# B&R Automation Studio project Panasonic_LinkaPowerCP2_A2021055 (part 30)

#### Main.st - Init, cyclic, exit code
```iecst
PROGRAM _INIT
	(* Insert code here *)

END_PROGRAM

PROGRAM _CYCLIC

	//**********************************************************IO modul Wedmuller**********************************************************************//
	//************Karta AB 3.5 8DI**************//
	P3_Pracovisko.IN.StavPrepatovejOchrany_OK := P3_Pracovisko.COM_Weidmuller.AB3_5_8DI.0;
	P3_Srobovanie.IN.NapajanieSkrutkovackyK40_OK := P3_Pracovisko.COM_Weidmuller.AB3_5_8DI.1;
	P3_Srobovanie.IN.NapajanieSkrutkovackyM5_OK := P3_Pracovisko.COM_Weidmuller.AB3_5_8DI.2;
	P3_Srobovanie.IN.NapajanieZasobnikaK40_OK := P3_Pracovisko.COM_Weidmuller.AB3_5_8DI.3;
	P3_Srobovanie.IN.NapajanieZasobnikaM5_OK := P3_Pracovisko.COM_Weidmuller.AB3_5_8DI.4;
	P3_Srobovanie.IN.NapajanieVibrolistyM5_OK := P3_Pracovisko.COM_Weidmuller.AB3_5_8DI.5;
	P3_LeakageTestA.IN.NapajanieTestera_OK := P3_Pracovisko.COM_Weidmuller.AB3_5_8DI.6;
	P3_LeakageTestB.IN.NapajanieTestera_OK := P3_Pracovisko.COM_Weidmuller.AB3_5_8DI.7;

	//************Karta AB 3.6 8DI**************//
	P3_Dopravniky.IN.StavRiadPredDopravBunky_READY := P3_Pracovisko.COM_Weidmuller.AB3_6_8DI.0;
	P3_Dopravniky.IN.StavRiadeniaPriecnDoprav1_READY := P3_Pracovisko.COM_Weidmuller.AB3_6_8DI.1;
	P3_Dopravniky.IN.StavRiadeniaPriecnDoprav2_READY := P3_Pracovisko.COM_Weidmuller.AB3_6_8DI.2;
	P3_Dopravniky.IN.StavRiadZadnDopravBunky_READY := P3_Pracovisko.COM_Weidmuller.AB3_6_8DI.3;
	P3_Dopravniky.IN.StavRiadeniaVratnehoDoprav_READY := P3_Pracovisko.COM_Weidmuller.AB3_6_8DI.4;
	P3_Dopravniky.IN.TeplotaMotoraPredDopravBunky_OK := P3_Pracovisko.COM_Weidmuller.AB3_6_8DI.5;
	P3_Dopravniky.IN.TeplotaMotoraPriecnDoprav1_OK := P3_Pracovisko.COM_Weidmuller.AB3_6_8DI.6;
	P3_Dopravniky.IN.TeplotaMotoraPriecnDoprav2_OK := P3_Pracovisko.COM_Weidmuller.AB3_6_8DI.7;

	//************Karta AB 3.7 8DI**************//
	P3_Dopravniky.IN.TeplotaMotoraZadnDopravBunky_OK := P3_Pracovisko.COM_Weidmuller.AB3_7_8DI.0;
	P3_Dopravniky.IN.TeplotaMotoraVratnehoDoprav_OK := P3_Pracovisko.COM_Weidmuller.AB3_7_8DI.1;
	P3_Pracovisko.COM_Weidmuller.AB3_7_8DI.2;
	P3_Pracovisko.COM_Weidmuller.AB3_7_8DI.3;
	Safety.IN.Linka_SV_ZonaCS := P3_Pracovisko.COM_Weidmuller.AB3_7_8DI.4;
	Safety.IN.P3_SV_ZonaBunky := P3_Pracovisko.COM_Weidmuller.AB3_7_8DI.5;
	Safety.IN.P3_SV_HV_test := P3_Pracovisko.COM_Weidmuller.AB3_7_8DI.6;
	P3_Pracovisko.COM_Weidmuller.AB3_7_8DI.7;

	//************Karta AB 3.8 8DI**************//
	P3_Pracovisko.COM_Weidmuller.AB3_8_8DI.0;
	P3_Pracovisko.COM_Weidmuller.AB3_8_8DI.1;
	P3_Pracovisko.COM_Weidmuller.AB3_8_8DI.2;
	P3_Pracovisko.COM_Weidmuller.AB3_8_8DI.3;
	P3_Pracovisko.COM_Weidmuller.AB3_8_8DI.4;
	P3_Pracovisko.COM_Weidmuller.AB3_8_8DI.5;
	P3_Pracovisko.COM_Weidmuller.AB3_8_8DI.6;
	P3_Pracovisko.COM_Weidmuller.AB3_8_8DI.7;

	//************Karta AB 3.9 8DO***************//
	P3_Pracovisko.COM_Weidmuller.AB3_9_8DO.0 := P3_Pracovisko.OUT.Majak_ZeleneSvetlo_ON;
	P3_Pracovisko.COM_Weidmuller.AB3_9_8DO.1 := P3_Pracovisko.OUT.Majak_OranzoveSvetlo_ON;
	P3_Pracovisko.COM_Weidmuller.AB3_9_8DO.2 := P3_Pracovisko.OUT.Majak_CerveneSvetlo_ON;
	P3_Pracovisko.COM_Weidmuller.AB3_9_8DO.3 := P3_Pracovisko.OUT.Majak_Hukacka_ON;
	P3_Pracovisko.COM_Weidmuller.AB3_9_8DO.4 := P3_Srobovanie.SkrutSet_K40.OUT.VibracnyHrniec.ZapniVibromotor;
	P3_Pracovisko.COM_Weidmuller.AB3_9_8DO.5 := P3_Srobovanie.SkrutSet_M5.OUT.VibropohonZasobnika_RUN;
	P3_Pracovisko.COM_Weidmuller.AB3_9_8DO.6 := P3_Srobovanie.SkrutSet_M5.OUT.VibropohonListy_RUN;
	P3_Pracovisko.COM_Weidmuller.AB3_9_8DO.7 := P3_Pracovisko.OUT.OsvetlenieBunky_ON;

	//************Karta AB 3.10 8DO***************//
	P3_Pracovisko.COM_Weidmuller.AB3_10_8DO.0;
	P3_Pracovisko.COM_Weidmuller.AB3_10_8DO.1;
	P3_Pracovisko.COM_Weidmuller.AB3_10_8DO.2;
	P3_Pracovisko.COM_Weidmuller.AB3_10_8DO.3;
	P3_Pracovisko.COM_Weidmuller.AB3_10_8DO.4;
	P3_Pracovisko.COM_Weidmuller.AB3_10_8DO.5:= Safety.OUT.Linka_ResetCS;
	P3_Pracovisko.COM_Weidmuller.AB3_10_8DO.6:= Safety.OUT.P3_ResetZonyBunky;
	P3_Pracovisko.COM_Weidmuller.AB3_10_8DO.7:= Safety.OUT.P3_ResetZonyHVtest;

	P3_Pracovisko.COM_Weidmuller.AB3_10_8DO.0 := P3_Dopravniky.OUT.PrednyDopravnikBunky_ON;
	P3_Pracovisko.COM_Weidmuller.AB3_10_8DO.1 := P3_Dopravniky.OUT.PriecnyDopravnik1_VPRED;
	P3_Pracovisko.COM_Weidmuller.AB3_10_8DO.2 := P3_Dopravniky.OUT.PriecnyDopravnik2_VPRED;
	P3_Pracovisko.COM_Weidmuller.AB3_10_8DO.3 := P3_Dopravniky.OUT.ZadnyDopravnikBunky_ON;
	P3_Pracovisko.COM_Weidmuller.AB3_10_8DO.4 := P3_Dopravniky.OUT.VratnyDopravnik_ON;
	P3_Pracovisko.COM_Weidmuller.AB3_10_8DO.5;
	P3_Pracovisko.COM_Weidmuller.AB3_10_8DO.6;
	P3_Pracovisko.COM_Weidmuller.AB3_10_8DO.7;

	//************Karta AB 3.12 8DO***************//
	P3_Pracovisko.COM_Weidmuller.AB3_12_8DO.0;
	P3_Pracovisko.COM_Weidmuller.AB3_12_8DO.1;
	P3_Pracovisko.COM_Weidmuller.AB3_12_8DO.2;
	P3_Pracovisko.COM_Weidmuller.AB3_12_8DO.3;
	P3_Pracovisko.COM_Weidmuller.AB3_12_8DO.4;
	P3_Pracovisko.COM_Weidmuller.AB3_12_8DO.5;
	P3_Pracovisko.COM_Weidmuller.AB3_12_8DO.6 := P3_Dopravniky.OUT.PriecnyDopravnik2_VZAD;
	P3_Pracovisko.COM_Weidmuller.AB3_12_8DO.7 := P3_Pracovisko.OUT.Ventilator_ON;

	//**************************************************************IO modul Festo**********************************************************************************//

	//**********Modul DM 3.1 4DI4DO**************//
	//Inputs//
	P3_Pracovisko.IN.PredneDvereLave_PritomnAdaptera := P3_Pracovisko.COM_Festo.DM3_1_4DI[0];
	P3_Pracovisko.IN.PredneDverePrave_PritomnAdaptera := P3_Pracovisko.COM_Festo.DM3_1_4DI[1];
	P3_Pracovisko.IN.ZadneDvereLave_PritomnAdaptera := P3_Pracovisko.COM_Festo.DM3_1_4DI[2];
	P3_Pracovisko.IN.ZadneDverePrave_PritomnAdaptera := P3_Pracovisko.COM_Festo.DM3_1_4DI[3];

	//Outputs//
	P3_Pracovisko.COM_Festo.DM3_1_4DO[0] := P3_Pracovisko.OUT.PredneDvereLave_ZAMKNI;
	P3_Pracovisko.COM_Festo.DM3_1_4DO[1] := P3_Pracovisko.OUT.PredneDverePrave_ZAMKNI;
	P3_Pracovisko.COM_Festo.DM3_1_4DO[2] := P3_Pracovisko.OUT.ZadneDvereLave_ZAMKNI;
	P3_Pracovisko.COM_Festo.DM3_1_4DO[3] := P3_Pracovisko.OUT.ZadneDverePrave_ZAMKNI;

	//***********Modul DI 3.1 8DI****************//
	P3_HV_Test.IN.HorneKontakty_VYSUNUTE := P3_Pracovisko.COM_Festo.DI3_1_8DI[0];
	P3_HV_Test.IN.HorneKontakty_ZASUNUTE := P3_Pracovisko.COM_Festo.DI3_1_8DI[1];
	P3_HV_Test.IN.Centrovanie_ZASUNUTE := P3_Pracovisko.COM_Festo.DI3_1_8DI[2];
	P3_HV_Test.IN.Centrovanie_VYSUNUTE := P3_Pracovisko.COM_Festo.DI3_1_8DI[3];
	P3_HV_Test.IN.SpodneKontakty_ZASUNUTE := P3_Pracovisko.COM_Festo.DI3_1_8DI[4];
	P3_HV_Test.IN.SpodneKontakty_VYSUNUTE := P3_Pracovisko.COM_Festo.DI3_1_8DI[5];
	P3_HV_Test.IN.TypKonektoru_5F_5H := P3_Pracovisko.COM_Festo.DI3_1_8DI[6];
	P3_HV_Test.IN.TypKonektoru_4F := P3_Pracovisko.COM_Festo.DI3_1_8DI[7];

	//***********Modul DI 3.2 8DI****************//
	P3_Pracovisko.COM_Festo.DI3_2_8DI[0];
	P3_ZdvizkaZaLeakTestA.IN.TlmicPaletky_ZASUNUTY := P3_Pracovisko.COM_Festo.DI3_2_8DI[1];
	P3_ZdvizkaZaLeakTestB.IN.TlmicPaletky_ZASUNUTY := P3_Pracovisko.COM_Festo.DI3_2_8DI[2];
	P3_Pracovisko.COM_Festo.DI3_2_8DI[3];
	P3_Pracovisko.COM_Festo.DI3_2_8DI[4];
	P3_Pracovisko.COM_Festo.DI3_2_8DI[5];
	P3_Pracovisko.COM_Festo.DI3_2_8DI[6];
	P3_Pracovisko.COM_Festo.DI3_2_8DI[7];

	//***********Modul DI 3.3 8DI****************//
	P3_LeakageTestA.IN.HornyPritlak_TlakOK := P3_Pracovisko.COM_Festo.DI3_4_8DI[0];
	P3_LeakageTestA.IN.HornyPritlak_PneuZamok_Odomknuty := P3_Pracovisko.COM_Festo.DI3_4_8DI[1];
	P3_LeakageTestB.IN.HornyPritlak_ZASUNUTY := P3_Pracovisko.COM_Festo.DI3_3_8DI[2];
	P3_LeakageTestB.IN.HornyPritlak_VYSUNUTY := P3_Pracovisko.COM_Festo.DI3_3_8DI[3];
	P3_LeakageTestB.IN.PritomnostKopita := P3_Pracovisko.COM_Festo.DI3_3_8DI[4];
	P3_LeakageTestB.IN.Kopito_ZASUNUTE := P3_Pracovisko.COM_Festo.DI3_3_8DI[5];
	P3_LeakageTestB.IN.Centrovanie_VYSUNUTE := P3_Pracovisko.COM_Festo.DI3_3_8DI[6];
	P3_LeakageTestB.IN.Centrovanie_ZASUNUTE := P3_Pracovisko.COM_Festo.DI3_3_8DI[7];

	//***********Modul DI 3.4 8DI****************//
	P3_LeakageTestB.IN.HornyPritlak_TlakOK:= P3_Pracovisko.COM_Festo.DI3_3_8DI[0];
	P3_LeakageTestB.IN.HornyPritlak_PneuZamok_Odomknuty := P3_Pracovisko.COM_Festo.DI3_3_8DI[1];
	P3_LeakageTestA.IN.HornyPritlak_VYSUNUTY := P3_Pracovisko.COM_Festo.DI3_4_8DI[2];
	P3_LeakageTestA.IN.HornyPritlak_ZASUNUTY := P3_Pracovisko.COM_Festo.DI3_4_8DI[3];
	P3_LeakageTestA.IN.PritomnostKopita := P3_Pracovisko.COM_Festo.DI3_4_8DI[4];
	P3_LeakageTestA.IN.Kopito_ZASUNUTE := P3_Pracovisko.COM_Festo.DI3_4_8DI[5];
	P3_LeakageTestA.IN.Centrovanie_VYSUNUTE := P3_Pracovisko.COM_Festo.DI3_4_8DI[6];
	P3_LeakageTestA.IN.Centrovanie_ZASUNUTE := P3_Pracovisko.COM_Festo.DI3_4_8DI[7];

	//***********Modul DI 3.5 8DI****************//
	P3_Srobovanie.SkrutSet_K40.IN.VibracnyHrniec.PritomnostSkrutiekVHrnci := P3_Pracovisko.COM_Festo.DI3_5_8DI[0];
	P3_Srobovanie.SkrutSet_K40.IN.VibracnyHrniec.VibracnaListaZaplnena := P3_Pracovisko.COM_Festo.DI3_5_8DI[1];
	P3_Srobovanie.SkrutSet_K40.IN.VibracnyHrniec.PreletovySnimac := P3_Pracovisko.COM_Festo.DI3_5_8DI[2];
	P3_Srobovanie.SkrutSet_K40.IN.Brzda.PodajSkrutku:= P3_Pracovisko.COM_Festo.DI3_5_8DI[3];
	P3_Srobovanie.SkrutSet_K40.IN.Brzda.ZakladnaPoloha  := P3_Pracovisko.COM_Festo.DI3_5_8DI[4];
	P3_Srobovanie.SkrutSet_K40.IN.Brzda.SkrutkaPritomnaVBrzde := P3_Pracovisko.COM_Festo.DI3_5_8DI[5];
	P3_Srobovanie.SkrutSet_K40.IN.Brzda.PreletSkrutky := P3_Pracovisko.COM_Festo.DI3_5_8DI[6];
	P3_Srobovanie.IN.Skrutkovacka_K40_ZASUNUTA := P3_Pracovisko.COM_Festo.DI3_5_8DI[7];

	//***********Modul DI 3.6 8DI****************//
	P3_Srobovanie.SkrutSet_M5.IN.ZasobnikSkrutiekPrazdny := P3_Pracovisko.COM_Festo.DI3_6_8DI[0];
	P3_Srobovanie.SkrutSet_M5.IN.ZaplnenieListyZasobnika := P3_Pracovisko.COM_Festo.DI3_6_8DI[1];
	P3_Srobovanie.SkrutSet_M5.IN.ZaplnenieVibrolisty_MAX := P3_Pracovisko.COM_Festo.DI3_6_8DI[2];
	P3_Srobovanie.SkrutSet_M5.IN.ZaplnenieVibrolisty_MIN := P3_Pracovisko.COM_Festo.DI3_6_8DI[3];
	P3_Srobovanie.SkrutSet_M5.IN.Podavac_SkrutkaNaVstupe := P3_Pracovisko.COM_Festo.DI3_6_8DI[4];
	P3_Srobovanie.SkrutSet_M5.IN.Podavac_SkrutkaNaVystupe := P3_Pracovisko.COM_Festo.DI3_6_8DI[5];
	P3_Srobovanie.SkrutSet_M5.IN.PodavacOtoceny_VSTUP := P3_Pracovisko.COM_Festo.DI3_6_8DI[6];
	P3_Srobovanie.SkrutSet_M5.IN.PodavacOtoceny_VYSTUP := P3_Pracovisko.COM_Festo.DI3_6_8DI[7];

	//***********Modul DI 3.7 8DI****************//
	P3_Srobovanie.IN.Skrutkovacka_M5_Vakum_OK := P3_Pracovisko.COM_Festo.DI3_7_8DI[0];
	P3_Pracovisko.IN.TlakVzduchu_OK := P3_Pracovisko.COM_Festo.DI3_7_8DI[1];
	Safety.IN.P3_SV_PrivodVzduchu_CH1 := P3_Pracovisko.COM_Festo.DI3_7_8DI[2];
	Safety.IN.P3_SV_PrivodVzduchu_CH2 := P3_Pracovisko.COM_Festo.DI3_7_8DI[3];
	P3_LeakageTestA.IN.Tester_TypKonektoru_4F:= P3_Pracovisko.COM_Festo.DI3_7_8DI[4];
	P3_LeakageTestA.IN.Tester_TypKonektoru_5F_5H:= P3_Pracovisko.COM_Festo.DI3_7_8DI[5];
	P3_LeakageTestB.IN.Tester_TypKonektoru_4F:= P3_Pracovisko.COM_Festo.DI3_7_8DI[6];
	P3_LeakageTestB.IN.Tester_TypKonektoru_5F_5H:= P3_Pracovisko.COM_Festo.DI3_7_8DI[7];

	//***********Modul DI 3.8 8DI****************//
	P3_ZdvizkaPredLeakTestA.IN.Zdvizka_HornaPoloha := P3_Pracovisko.COM_Festo.DI3_8_8DI[0];
	P3_ZdvizkaPredLeakTestA.IN.Zdvizka_SpodnaPoloha := P3_Pracovisko.COM_Festo.DI3_8_8DI[1];
	P3_ZdvizkaPredLeakTestA.IN.Zdvizka_StrednaPoloha := P3_Pracovisko.COM_Festo.DI3_8_8DI[2];
	P3_ZdvizkaPredLeakTestA.IN.PritomnostPaletky := P3_Pracovisko.COM_Festo.DI3_8_8DI[3];
	P3_ZdvizkaPredLeakTestB.IN.Zdvizka_SpodnaPoloha := P3_Pracovisko.COM_Festo.DI3_8_8DI[4];
	P3_ZdvizkaPredLeakTestB.IN.Zdvizka_HornaPoloha := P3_Pracovisko.COM_Festo.DI3_8_8DI[5];
	P3_ZdvizkaPredLeakTestB.IN.Zdvizka_StrednaPoloha := P3_Pracovisko.COM_Festo.DI3_8_8DI[6];
	P3_ZdvizkaPredLeakTestB.IN.PoziciaPaletky_OK := P3_Pracovisko.COM_Festo.DI3_8_8DI[7];

	//***********Modul DI 3.9 8DI****************//
	P3_ZdvizkaPredLeakTestB.IN.PritomnostPaletky := P3_Pracovisko.COM_Festo.DI3_9_8DI[0];
	P3_ZdvizkaZaLeakTestA.IN.Zdvizka_SpodnaPoloha := P3_Pracovisko.COM_Festo.DI3_9_8DI[1];
	P3_ZdvizkaZaLeakTestA.IN.Zdvizka_HornaPoloha := P3_Pracovisko.COM_Festo.DI3_9_8DI[2];
	P3_ZdvizkaZaLeakTestA.IN.Zdvizka_StrednaPoloha := P3_Pracovisko.COM_Festo.DI3_9_8DI[3];
	P3_ZdvizkaZaLeakTestA.IN.PritomnostPaletky := P3_Pracovisko.COM_Festo.DI3_9_8DI[4];
	P3_ZdvizkaZaLeakTestA.IN.PoziciaPaletky_OK := P3_Pracovisko.COM_Festo.DI3_9_8DI[5];
	P3_SpodnyStoper.IN.ZaplnenieDopravnika := P3_Pracovisko.COM_Festo.DI3_9_8DI[6];
	P3_SpodnyStoper.IN.PritomnostPaletky := P3_Pracovisko.COM_Festo.DI3_9_8DI[7];

	//***********Modul DI 3.10 8DI****************//
	P3_ZdvizkaZaLeakTestB.IN.Zdvizka_SpodnaPoloha := P3_Pracovisko.COM_Festo.DI3_10_8DI[0];
	P3_ZdvizkaZaLeakTestB.IN.Zdvizka_HornaPoloha  := P3_Pracovisko.COM_Festo.DI3_10_8DI[1];
	P3_ZdvizkaZaLeakTestB.IN.Zdvizka_StrednaPoloha := P3_Pracovisko.COM_Festo.DI3_10_8DI[2];
	P3_ZdvizkaZaLeakTestB.IN.PritomnostPaletky := P3_Pracovisko.COM_Festo.DI3_10_8DI[3];
	P3_ZdvizkaZaLeakTestB.IN.PoziciaPaletky_OK := P3_Pracovisko.COM_Festo.DI3_10_8DI[4];
	P3_Pracovisko.COM_Festo.DI3_10_8DI[5];
	P3_StoperSrobovania.IN.Centrovanie_VYSUNUTE:= P3_Pracovisko.COM_Festo.DI3_10_8DI[6];
	P3_StoperSrobovania.IN.Centrovanie_ZASUNUTE := P3_Pracovisko.COM_Festo.DI3_10_8DI[7];

	//********Modul DS 3.1 IO link Port 0 - RFID snímač paletky stoper skrutkovania**************//
	//Inputs//
	P3_StoperSrobovania.RFID_hlava.Mapping_IN[0]:= P3_Pracovisko.COM_Festo.DS3_1_Port0_IN[0];
	P3_StoperSrobovania.RFID_hlava.Mapping_IN[1]:= P3_Pracovisko.COM_Festo.DS3_1_Port0_IN[1];
	P3_StoperSrobovania.RFID_hlava.Mapping_IN[2]:= P3_Pracovisko.COM_Festo.DS3_1_Port0_IN[2];
	P3_StoperSrobovania.RFID_hlava.Mapping_IN[3]:= P3_Pracovisko.COM_Festo.DS3_1_Port0_IN[3];
	P3_StoperSrobovania.RFID_hlava.Mapping_IN[4]:= P3_Pracovisko.COM_Festo.DS3_1_Port0_IN[4];
	P3_StoperSrobovania.RFID_hlava.Mapping_IN[5]:= P3_Pracovisko.COM_Festo.DS3_1_Port0_IN[5];
	P3_StoperSrobovania.RFID_hlava.Mapping_IN[6]:= P3_Pracovisko.COM_Festo.DS3_1_Port0_IN[6];
	P3_StoperSrobovania.RFID_hlava.Mapping_IN[7]:= P3_Pracovisko.COM_Festo.DS3_1_Port0_IN[7];

	//Outputs//
	P3_Pracovisko.COM_Festo.DS3_1_Port0_OUT[0]:= P3_StoperSrobovania.RFID_hlava.Mapping_OUT[0];
	P3_Pracovisko.COM_Festo.DS3_1_Port0_OUT[1]:= P3_StoperSrobovania.RFID_hlava.Mapping_OUT[1];
	P3_Pracovisko.COM_Festo.DS3_1_Port0_OUT[2]:= P3_StoperSrobovania.RFID_hlava.Mapping_OUT[2];
	P3_Pracovisko.COM_Festo.DS3_1_Port0_OUT[3]:= P3_StoperSrobovania.RFID_hlava.Mapping_OUT[3];
	P3_Pracovisko.COM_Festo.DS3_1_Port0_OUT[4]:= P3_StoperSrobovania.RFID_hlava.Mapping_OUT[4];
	P3_Pracovisko.COM_Festo.DS3_1_Port0_OUT[5]:= P3_StoperSrobovania.RFID_hlava.Mapping_OUT[5];
	P3_Pracovisko.COM_Festo.DS3_1_Port0_OUT[6]:= P3_StoperSrobovania.RFID_hlava.Mapping_OUT[6];
	P3_Pracovisko.COM_Festo.DS3_1_Port0_OUT[7]:= P3_StoperSrobovania.RFID_hlava.Mapping_OUT[7];

	//********Modul DS 3.1 IO link Port 1 - RFID snímač paletky HV test**************//
	//Inputs//
	P3_HV_Test.RFID_hlava.Mapping_IN[0]:= P3_Pracovisko.COM_Festo.DS3_1_Port1_IN[0];
	P3_HV_Test.RFID_hlava.Mapping_IN[1]:= P3_Pracovisko.COM_Festo.DS3_1_Port1_IN[1];
	P3_HV_Test.RFID_hlava.Mapping_IN[2]:= P3_Pracovisko.COM_Festo.DS3_1_Port1_IN[2];
	P3_HV_Test.RFID_hlava.Mapping_IN[3]:= P3_Pracovisko.COM_Festo.DS3_1_Port1_IN[3];
	P3_HV_Test.RFID_hlava.Mapping_IN[4]:= P3_Pracovisko.COM_Festo.DS3_1_Port1_IN[4];
	P3_HV_Test.RFID_hlava.Mapping_IN[5]:= P3_Pracovisko.COM_Festo.DS3_1_Port1_IN[5];
	P3_HV_Test.RFID_hlava.Mapping_IN[6]:= P3_Pracovisko.COM_Festo.DS3_1_Port1_IN[6];
	P3_HV_Test.RFID_hlava.Mapping_IN[7]:= P3_Pracovisko.COM_Festo.DS3_1_Port1_IN[7];

	//Outputs//
	P3_Pracovisko.COM_Festo.DS3_1_Port1_OUT[0]:= P3_HV_Test.RFID_hlava.Mapping_OUT[0];
	P3_Pracovisko.COM_Festo.DS3_1_Port1_OUT[1]:= P3_HV_Test.RFID_hlava.Mapping_OUT[1];
	P3_Pracovisko.COM_Festo.DS3_1_Port1_OUT[2]:= P3_HV_Test.RFID_hlava.Mapping_OUT[2];
	P3_Pracovisko.COM_Festo.DS3_1_Port1_OUT[3]:= P3_HV_Test.RFID_hlava.Mapping_OUT[3];
	P3_Pracovisko.COM_Festo.DS3_1_Port1_OUT[4]:= P3_HV_Test.RFID_hlava.Mapping_OUT[4];
	P3_Pracovisko.COM_Festo.DS3_1_Port1_OUT[5]:= P3_HV_Test.RFID_hlava.Mapping_OUT[5];
	P3_Pracovisko.COM_Festo.DS3_1_Port1_OUT[6]:= P3_HV_Test.RFID_hlava.Mapping_OUT[6];
	P3_Pracovisko.COM_Festo.DS3_1_Port1_OUT[7]:= P3_HV_Test.RFID_hlava.Mapping_OUT[7];

	//********Modul DS 3.1 IO link Port 2 - RFID snímač paletky Leakage test B**************//
	//Inputs//
	P3_LeakageTestB.RFID_hlava.Mapping_IN[0]:= P3_Pracovisko.COM_Festo.DS3_1_Port2_IN[0];
	P3_LeakageTestB.RFID_hlava.Mapping_IN[1]:= P3_Pracovisko.COM_Festo.DS3_1_Port2_IN[1];
	P3_LeakageTestB.RFID_hlava.Mapping_IN[2]:= P3_Pracovisko.COM_Festo.DS3_1_Port2_IN[2];
	P3_LeakageTestB.RFID_hlava.Mapping_IN[3]:= P3_Pracovisko.COM_Festo.DS3_1_Port2_IN[3];
	P3_LeakageTestB.RFID_hlava.Mapping_IN[4]:= P3_Pracovisko.COM_Festo.DS3_1_Port2_IN[4];
	P3_LeakageTestB.RFID_hlava.Mapping_IN[5]:= P3_Pracovisko.COM_Festo.DS3_1_Port2_IN[5];
	P3_LeakageTestB.RFID_hlava.Mapping_IN[6]:= P3_Pracovisko.COM_Festo.DS3_1_Port2_IN[6];
	P3_LeakageTestB.RFID_hlava.Mapping_IN[7]:= P3_Pracovisko.COM_Festo.DS3_1_Port2_IN[7];

	//Outputs//
	P3_Pracovisko.COM_Festo.DS3_1_Port2_OUT[0]:= P3_LeakageTestB.RFID_hlava.Mapping_OUT[0];
	P3_Pracovisko.COM_Festo.DS3_1_Port2_OUT[1]:= P3_LeakageTestB.RFID_hlava.Mapping_OUT[1];
	P3_Pracovisko.COM_Festo.DS3_1_Port2_OUT[2]:= P3_LeakageTestB.RFID_hlava.Mapping_OUT[2];
	P3_Pracovisko.COM_Festo.DS3_1_Port2_OUT[3]:= P3_LeakageTestB.RFID_hlava.Mapping_OUT[3];
	P3_Pracovisko.COM_Festo.DS3_1_Port2_OUT[4]:= P3_LeakageTestB.RFID_hlava.Mapping_OUT[4];
	P3_Pracovisko.COM_Festo.DS3_1_Port2_OUT[5]:= P3_LeakageTestB.RFID_hlava.Mapping_OUT[5];
	P3_Pracovisko.COM_Festo.DS3_1_Port2_OUT[6]:= P3_LeakageTestB.RFID_hlava.Mapping_OUT[6];
	P3_Pracovisko.COM_Festo.DS3_1_Port2_OUT[7]:= P3_LeakageTestB.RFID_hlava.Mapping_OUT[7];

	//********Modul DS 3.1 IO link Port 3 - RFID snímač paletky Leakage test A**************//
	//Inputs//
	P3_LeakageTestA.RFID_hlava.Mapping_IN[0]:= P3_Pracovisko.COM_Festo.DS3_1_Port3_IN[0];
	P3_LeakageTestA.RFID_hlava.Mapping_IN[1]:= P3_Pracovisko.COM_Festo.DS3_1_Port3_IN[1];
	P3_LeakageTestA.RFID_hlava.Mapping_IN[2]:= P3_Pracovisko.COM_Festo.DS3_1_Port3_IN[2];
	P3_LeakageTestA.RFID_hlava.Mapping_IN[3]:= P3_Pracovisko.COM_Festo.DS3_1_Port3_IN[3];
	P3_LeakageTestA.RFID_hlava.Mapping_IN[4]:= P3_Pracovisko.COM_Festo.DS3_1_Port3_IN[4];
	P3_LeakageTestA.RFID_hlava.Mapping_IN[5]:= P3_Pracovisko.COM_Festo.DS3_1_Port3_IN[5];
	P3_LeakageTestA.RFID_hlava.Mapping_IN[6]:= P3_Pracovisko.COM_Festo.DS3_1_Port3_IN[6];
	P3_LeakageTestA.RFID_hlava.Mapping_IN[7]:= P3_Pracovisko.COM_Festo.DS3_1_Port3_IN[7];

	//Outputs//
	P3_Pracovisko.COM_Festo.DS3_1_Port3_OUT[0]:= P3_LeakageTestA.RFID_hlava.Mapping_OUT[0];
	P3_Pracovisko.COM_Festo.DS3_1_Port3_OUT[1]:= P3_LeakageTestA.RFID_hlava.Mapping_OUT[1];
	P3_Pracovisko.COM_Festo.DS3_1_Port3_OUT[2]:= P3_LeakageTestA.RFID_hlava.Mapping_OUT[2];
	P3_Pracovisko.COM_Festo.DS3_1_Port3_OUT[3]:= P3_LeakageTestA.RFID_hlava.Mapping_OUT[3];
	P3_Pracovisko.COM_Festo.DS3_1_Port3_OUT[4]:= P3_LeakageTestA.RFID_hlava.Mapping_OUT[4];
	P3_Pracovisko.COM_Festo.DS3_1_Port3_OUT[5]:= P3_LeakageTestA.RFID_hlava.Mapping_OUT[5];
	P3_Pracovisko.COM_Festo.DS3_1_Port3_OUT[6]:= P3_LeakageTestA.RFID_hlava.Mapping_OUT[6];
	P3_Pracovisko.COM_Festo.DS3_1_Port3_OUT[7]:= P3_LeakageTestA.RFID_hlava.Mapping_OUT[7];

	//*********Modul DS 3.2 IO link Port 0 - Snímač tlaku Leakage test B****************//
	//Inputs//
	P3_Pracovisko.COM_Festo.DS3_2_Port0_IN[0];
	P3_Pracovisko.COM_Festo.DS3_2_Port0_IN[1];

	P3_LeakageTestB.IN.VyrovnavaciTlak_OK:= P3_Pracovisko.COM_Festo.DS3_2_Port0_IN[1].0;

	P3_LeakageTestB.PAR.PrecitanyVyrovnavaciTlak.0:= P3_Pracovisko.COM_Festo.DS3_2_Port0_IN[1].2;
	P3_LeakageTestB.PAR.PrecitanyVyrovnavaciTlak.1:= P3_Pracovisko.COM_Festo.DS3_2_Port0_IN[1].3;
	P3_LeakageTestB.PAR.PrecitanyVyrovnavaciTlak.2:= P3_Pracovisko.COM_Festo.DS3_2_Port0_IN[1].4;
	P3_LeakageTestB.PAR.PrecitanyVyrovnavaciTlak.3:= P3_Pracovisko.COM_Festo.DS3_2_Port0_IN[1].5;
	P3_LeakageTestB.PAR.PrecitanyVyrovnavaciTlak.4:= P3_Pracovisko.COM_Festo.DS3_2_Port0_IN[1].6;
	P3_LeakageTestB.PAR.PrecitanyVyrovnavaciTlak.5:= P3_Pracovisko.COM_Festo.DS3_2_Port0_IN[1].7;
	P3_LeakageTestB.PAR.PrecitanyVyrovnavaciTlak.6:= P3_Pracovisko.COM_Festo.DS3_2_Port0_IN[0].0;
	P3_LeakageTestB.PAR.PrecitanyVyrovnavaciTlak.7:= P3_Pracovisko.COM_Festo.DS3_2_Port0_IN[0].1;
	P3_LeakageTestB.PAR.PrecitanyVyrovnavaciTlak.8:= P3_Pracovisko.COM_Festo.DS3_2_Port0_IN[0].2;
	P3_LeakageTestB.PAR.PrecitanyVyrovnavaciTlak.9:= P3_Pracovisko.COM_Festo.DS3_2_Port0_IN[0].3;
	P3_LeakageTestB.PAR.PrecitanyVyrovnavaciTlak.10:= P3_Pracovisko.COM_Festo.DS3_2_Port0_IN[0].4;
	P3_LeakageTestB.PAR.PrecitanyVyrovnavaciTlak.11:= P3_Pracovisko.COM_Festo.DS3_2_Port0_IN[0].5;
	P3_LeakageTestB.PAR.PrecitanyVyrovnavaciTlak.12:= P3_Pracovisko.COM_Festo.DS3_2_Port0_IN[0].6;
	P3_LeakageTestB.PAR.PrecitanyVyrovnavaciTlak.13:= P3_Pracovisko.COM_Festo.DS3_2_Port0_IN[0].7;

	P3_LeakageTestB.PAR.PreratanyVyrovnavaciTlak_Bar:= P3_LeakageTestB.PAR.PrecitanyVyrovnavaciTlak*0.1;

	//*********Modul DS 3.2 IO link Port 1 - Snímač tlaku Leakage test A****************//
	//Inputs//
	P3_Pracovisko.COM_Festo.DS3_2_Port1_IN[0];
	P3_Pracovisko.COM_Festo.DS3_2_Port1_IN[1];

	P3_LeakageTestA.IN.VyrovnavaciTlak_OK:= P3_Pracovisko.COM_Festo.DS3_2_Port1_IN[1].0;

	P3_LeakageTestA.PAR.PrecitanyVyrovnavaciTlak.0:= P3_Pracovisko.COM_Festo.DS3_2_Port1_IN[1].2;
	P3_LeakageTestA.PAR.PrecitanyVyrovnavaciTlak.1:= P3_Pracovisko.COM_Festo.DS3_2_Port1_IN[1].3;
	P3_LeakageTestA.PAR.PrecitanyVyrovnavaciTlak.2:= P3_Pracovisko.COM_Festo.DS3_2_Port1_IN[1].4;
	P3_LeakageTestA.PAR.PrecitanyVyrovnavaciTlak.3:= P3_Pracovisko.COM_Festo.DS3_2_Port1_IN[1].5;
	P3_LeakageTestA.PAR.PrecitanyVyrovnavaciTlak.4:= P3_Pracovisko.COM_Festo.DS3_2_Port1_IN[1].6;
	P3_LeakageTestA.PAR.PrecitanyVyrovnavaciTlak.5:= P3_Pracovisko.COM_Festo.DS3_2_Port1_IN[1].7;
	P3_LeakageTestA.PAR.PrecitanyVyrovnavaciTlak.6:= P3_Pracovisko.COM_Festo.DS3_2_Port1_IN[0].0;
	P3_LeakageTestA.PAR.PrecitanyVyrovnavaciTlak.7:= P3_Pracovisko.COM_Festo.DS3_2_Port1_IN[0].1;
	P3_LeakageTestA.PAR.PrecitanyVyrovnavaciTlak.8:= P3_Pracovisko.COM_Festo.DS3_2_Port1_IN[0].2;
	P3_LeakageTestA.PAR.PrecitanyVyrovnavaciTlak.9:= P3_Pracovisko.COM_Festo.DS3_2_Port1_IN[0].3;
	P3_LeakageTestA.PAR.PrecitanyVyrovnavaciTlak.10:= P3_Pracovisko.COM_Festo.DS3_2_Port1_IN[0].4;
	P3_LeakageTestA.PAR.PrecitanyVyrovnavaciTlak.11:= P3_Pracovisko.COM_Festo.DS3_2_Port1_IN[0].5;
	P3_LeakageTestA.PAR.PrecitanyVyrovnavaciTlak.12:= P3_Pracovisko.COM_Festo.DS3_2_Port1_IN[0].6;
	P3_LeakageTestA.PAR.PrecitanyVyrovnavaciTlak.13:= P3_Pracovisko.COM_Festo.DS3_2_Port1_IN[0].7;

	P3_LeakageTestA.PAR.PreratanyVyrovnavaciTlak_Bar:= P3_LeakageTestA.PAR.PrecitanyVyrovnavaciTlak*0.1;

	//*********Modul DS 3.2 IO link Port 2 - Snímač vysunutia skrutkovačky K40****************//
	//Inputs//
	Convert_0.IN_Byte1:= P3_Pracovisko.COM_Festo.DS3_2_Port2_IN[0];
	Convert_0.IN_Byte0:= P3_Pracovisko.COM_Festo.DS3_2_Port2_IN[1];

	P3_Srobovanie.PAR.Skrutkov_K40_AktualHodnVysunutia:= Convert_0.OUT_UINT;
	Convert_0();

	//************************************Ventilový terminál*******************************************//

	//0-7
	P3_Pracovisko.COM_VentilovyTerminal[0].0 := P3_Srobovanie.OUT.Skrutkovacka_M5_Prisavanie_ON;
	P3_Pracovisko.COM_VentilovyTerminal[0].1 := P3_Srobovanie.OUT.Skrutkovacka_M5_Prisavanie_OFF;
	P3_Pracovisko.COM_VentilovyTerminal[0].2 := P3_Srobovanie.OUT.Skrutkovacka_M5_Odvzdusn_ON;
	P3_Pracovisko.COM_VentilovyTerminal[0].3;
	P3_Pracovisko.COM_VentilovyTerminal[0].4;
	P3_Pracovisko.COM_VentilovyTerminal[0].5;
	P3_Pracovisko.COM_VentilovyTerminal[0].6 := P3_StoperSrobovania.OUT.ZasunStoper;
	P3_Pracovisko.COM_VentilovyTerminal[0].7 := P3_HV_Test.OUT.ZasunStoper;

	//8-15
	P3_Pracovisko.COM_VentilovyTerminal[1].0 := P3_ZdvizkaPredLeakTestA.OUT.Zdvizku_VYSUN;
	P3_Pracovisko.COM_VentilovyTerminal[1].1 := P3_ZdvizkaPredLeakTestA.OUT.Zdvizku_ZASUN;
	P3_Pracovisko.COM_VentilovyTerminal[1].2 := P3_ZdvizkaPredLeakTestA.OUT.TlmicPaletky_VYSUN;
	P3_Pracovisko.COM_VentilovyTerminal[1].3;
	P3_Pracovisko.COM_VentilovyTerminal[1].4 := P3_ZdvizkaPredLeakTestB.OUT.Zdvizku_VYSUN;
	P3_Pracovisko.COM_VentilovyTerminal[1].5 := P3_ZdvizkaPredLeakTestB.OUT.Zdvizku_ZASUN;
	P3_Pracovisko.COM_VentilovyTerminal[1].6;
	P3_Pracovisko.COM_VentilovyTerminal[1].7;

	//16-23
	P3_Pracovisko.COM_VentilovyTerminal[2].0 := P3_LeakageTestA.OUT.ZasunStoper;
	P3_Pracovisko.COM_VentilovyTerminal[2].1 := P3_LeakageTestB.OUT.ZasunStoper;
	P3_Pracovisko.COM_VentilovyTerminal[2].2 := P3_ZdvizkaZaLeakTestA.OUT.Zdvizku_VYSUN;
	P3_Pracovisko.COM_VentilovyTerminal[2].3 := P3_ZdvizkaZaLeakTestA.OUT.Zdvizku_ZASUN;
	P3_Pracovisko.COM_VentilovyTerminal[2].4 := P3_ZdvizkaZaLeakTestA.OUT.TlmicPaletky_VYSUN;
	P3_Pracovisko.COM_VentilovyTerminal[2].5 := P3_ZdvizkaZaLeakTestA.OUT.TlmicPaletky_ZASUN;
	P3_Pracovisko.COM_VentilovyTerminal[2].6 := P3_ZdvizkaZaLeakTestB.OUT.Zdvizku_VYSUN;
	P3_Pracovisko.COM_VentilovyTerminal[2].7 := P3_ZdvizkaZaLeakTestB.OUT.Zdvizku_ZASUN;

	//24-31
	P3_Pracovisko.COM_VentilovyTerminal[3].0 := P3_ZdvizkaZaLeakTestB.OUT.TlmicPaletky_VYSUN;
	P3_Pracovisko.COM_VentilovyTerminal[3].1 := P3_ZdvizkaZaLeakTestB.OUT.TlmicPaletky_ZASUN;
	P3_Pracovisko.COM_VentilovyTerminal[3].2 := P3_Pracovisko.OUT.ZdvizkyPneuZamok_ODOMKNI;
	P3_Pracovisko.COM_VentilovyTerminal[3].3 := P3_SpodnyStoper.OUT.ZasunStoper;
	P3_Pracovisko.COM_VentilovyTerminal[3].4 := P3_Srobovanie.SkrutSet_K40.OUT.VibracnyHrniec.PrerusenieZasobovaniaSkrutiek;
	P3_Pracovisko.COM_VentilovyTerminal[3].5 := P3_Srobovanie.SkrutSet_K40.OUT.VibracnyHrniec.TiedenieSkrutiek;
	P3_Pracovisko.COM_VentilovyTerminal[3].6 := P3_Srobovanie.SkrutSet_K40.OUT.VibracnyHrniec.OddelovacVysunut;
	P3_Pracovisko.COM_VentilovyTerminal[3].7;

	//32-39
	P3_Pracovisko.COM_VentilovyTerminal[4].0 := P3_Srobovanie.SkrutSet_K40.OUT.VibracnyHrniec.VzduchNastreleniaSkrutky;
	P3_Pracovisko.COM_VentilovyTerminal[4].1;
	P3_Pracovisko.COM_VentilovyTerminal[4].2 := P3_Srobovanie.OUT.Skrutkovacka_K40_Prisavanie_ON;
	P3_Pracovisko.COM_VentilovyTerminal[4].3 := P3_Srobovanie.OUT.Skrutkovacka_K40_Odvzdusn_ON;
	P3_Pracovisko.COM_VentilovyTerminal[4].4 := P3_Srobovanie.SkrutSet_K40.OUT.Brzda.PodajSkrutku;
	P3_Pracovisko.COM_VentilovyTerminal[4].5 := P3_Srobovanie.SkrutSet_K40.OUT.Brzda.ZakladnaPoloha;
	P3_Pracovisko.COM_VentilovyTerminal[4].6 := P3_Srobovanie.SkrutSet_K40.OUT.Brzda.OdsavanieNecistot;
	P3_Pracovisko.COM_VentilovyTerminal[4].7 := P3_Srobovanie.SkrutSet_K40.OUT.Brzda.NastrelenieSkrutky;

	//40-47
	P3_Pracovisko.COM_VentilovyTerminal[5].0 := P3_Srobovanie.SkrutSet_M5.OUT.ZhadzovaciVzduch_RUN;
	P3_Pracovisko.COM_VentilovyTerminal[5].1 := P3_Srobovanie.SkrutSet_M5.OUT.TriediaciVzduch_RUN;
	P3_Pracovisko.COM_VentilovyTerminal[5].2 := P3_Srobovanie.SkrutSet_M5.OUT.OtocPodavac_NaVystup;
	P3_Pracovisko.COM_VentilovyTerminal[5].3 := P3_Srobovanie.SkrutSet_M5.OUT.OtocPodavac_NaVstup;
	P3_Pracovisko.COM_VentilovyTerminal[5].4 := P3_HV_Test.OUT.PritlacenieKontaktovTestera_ON;
	P3_Pracovisko.COM_VentilovyTerminal[5].5;
	P3_Pracovisko.COM_VentilovyTerminal[5].6 := P3_StoperSrobovania.OUT.Centrovanie_VYSUN;
	P3_Pracovisko.COM_VentilovyTerminal[5].7 := P3_StoperSrobovania.OUT.Centrovanie_ZASUN;

	//48-55
	P3_Pracovisko.COM_VentilovyTerminal[6].0 := P3_Srobovanie.OUT.Skrutkovacku_K40_VYSUN;
	P3_Pracovisko.COM_VentilovyTerminal[6].1;
	P3_Pracovisko.COM_VentilovyTerminal[6].2 := P3_HV_Test.OUT.Centrovanie_VYSUN;
	P3_Pracovisko.COM_VentilovyTerminal[6].3 := P3_HV_Test.OUT.Centrovanie_ZASUN;
	P3_Pracovisko.COM_VentilovyTerminal[6].4 := P3_HV_Test.OUT.SpodneKontakty_VYSUN;
	P3_Pracovisko.COM_VentilovyTerminal[6].5 := P3_HV_Test.OUT.SpodneKontakty_ZASUN;
	P3_Pracovisko.COM_VentilovyTerminal[6].6 := P3_HV_Test.OUT.HorneKontakty_VYSUN;
	P3_Pracovisko.COM_VentilovyTerminal[6].7 := P3_HV_Test.OUT.HorneKontakty_ZASUN;

	//56-63
	P3_Pracovisko.COM_VentilovyTerminal[7].0 := P3_HV_Test.OUT.PruzenieHornychKontaktov_VYSUN;
	P3_Pracovisko.COM_VentilovyTerminal[7].1 := P3_HV_Test.OUT.PruzenieHornychKontaktov_ZASUN;
	P3_Pracovisko.COM_VentilovyTerminal[7].2;
	P3_Pracovisko.COM_VentilovyTerminal[7].3;
	P3_Pracovisko.COM_VentilovyTerminal[7].4;
	P3_Pracovisko.COM_VentilovyTerminal[7].5;
	P3_Pracovisko.COM_VentilovyTerminal[7].6 := P3_LeakageTestA.OUT.Kopito_VYSUN;
	P3_Pracovisko.COM_VentilovyTerminal[7].7 := P3_LeakageTestA.OUT.Kopito_ZASUN;

	//64-71
	P3_Pracovisko.COM_VentilovyTerminal[8].0 := P3_LeakageTestA.OUT.Centrovanie_VYSUN;
	P3_Pracovisko.COM_VentilovyTerminal[8].1;
	P3_Pracovisko.COM_VentilovyTerminal[8].2 := P3_LeakageTestA.OUT.PneuZamokCentrovania_ODOMKNI;
	P3_Pracovisko.COM_VentilovyTerminal[8].3 := P3_LeakageTestA.OUT.PneuZamokZvonu_ODOMKNI;
	P3_Pracovisko.COM_VentilovyTerminal[8].4 := P3_LeakageTestA.OUT.HornyPritlak_VYSUN;
	P3_Pracovisko.COM_VentilovyTerminal[8].5 := P3_LeakageTestA.OUT.HornyPritlak_ZASUN;
	P3_Pracovisko.COM_VentilovyTerminal[8].6 := P3_LeakageTestB.OUT.Kopito_VYSUN;
	P3_Pracovisko.COM_VentilovyTerminal[8].7 := P3_LeakageTestB.OUT.Kopito_ZASUN;

	//72-79
	P3_Pracovisko.COM_VentilovyTerminal[9].0 := P3_LeakageTestB.OUT.Centrovanie_VYSUN;
	P3_Pracovisko.COM_VentilovyTerminal[9].1;
	P3_Pracovisko.COM_VentilovyTerminal[9].2 := P3_LeakageTestB.OUT.PneuZamokCentrovania_ODOMKNI;
	P3_Pracovisko.COM_VentilovyTerminal[9].3 := P3_LeakageTestB.OUT.PneuZamokZvonu_ODOMKNI;
	P3_Pracovisko.COM_VentilovyTerminal[9].4 := P3_LeakageTestB.OUT.HornyPritlak_VYSUN;
	P3_Pracovisko.COM_VentilovyTerminal[9].5 := P3_LeakageTestB.OUT.HornyPritlak_ZASUN;
	P3_Pracovisko.COM_VentilovyTerminal[9].6;
	P3_Pracovisko.COM_VentilovyTerminal[9].7;

	//Volanie knižníc//
	P3_Srobovanie.SkrutSet_K40();
	P3_Srobovanie.SkrutSet_M5();
	P3_Srobovanie.ServoManipulOsY();
	P3_Srobovanie.ServoManipulOsZ_M5();

END_PROGRAM

PROGRAM _EXIT
	(* Insert code here *)

END_PROGRAM
```

#### Variables.var - Local variables
```iecst
VAR
	Convert_0 : UsintToUint := (0);
END_VAR
```

### Program Logical/Program/Pracovisko_3/P3_OvladSafety (IEC)

#### Main.st - Init, cyclic, exit code
```iecst
PROGRAM _INIT
	(* Insert code here *)

END_PROGRAM

PROGRAM _CYCLIC

	//******************************************Ovládanie zámkov dverí bunky****************************************//
	//Zadné dvere //
	IF P34_Vizu.TL_ZamkniZadneZamky_P3 THEN
		IF NOT P3_Pracovisko.STAV.ZadneDvereZamknute AND P3_Pracovisko.IN.ZadneDvereLave_PritomnAdaptera AND P3_Pracovisko.IN.ZadneDverePrave_PritomnAdaptera THEN
			P3_Pracovisko.OUT.ZadneDvereLave_ZAMKNI:= TRUE;
			P3_Pracovisko.OUT.ZadneDverePrave_ZAMKNI:= TRUE;
		ELSIF P3_Pracovisko.STAV.ZadneDvereZamknute THEN
			P3_Pracovisko.OUT.ZadneDvereLave_ZAMKNI:= FALSE;
			P3_Pracovisko.OUT.ZadneDverePrave_ZAMKNI:= FALSE;
		END_IF
		P34_Vizu.TL_ZamkniZadneZamky_P3:= FALSE;
	END_IF

	//Predné dvere //
	IF P34_Vizu.TL_ZamkniPredneZamky_P3 THEN
		IF NOT P3_Pracovisko.STAV.PredneDvereZamknute AND P3_Pracovisko.IN.PredneDvereLave_PritomnAdaptera AND P3_Pracovisko.IN.PredneDverePrave_PritomnAdaptera THEN
			P3_Pracovisko.OUT.PredneDvereLave_ZAMKNI:= TRUE;
			P3_Pracovisko.OUT.PredneDverePrave_ZAMKNI:= TRUE;
		ELSIF P3_Pracovisko.STAV.PredneDvereZamknute THEN
			P3_Pracovisko.OUT.PredneDvereLave_ZAMKNI:= FALSE;
			P3_Pracovisko.OUT.PredneDverePrave_ZAMKNI:= FALSE;
		END_IF
		P34_Vizu.TL_ZamkniPredneZamky_P3:= FALSE;
	END_IF

	//Stav zadné dvere zamknuté//
	IF P3_Pracovisko.OUT.ZadneDvereLave_ZAMKNI AND P3_Pracovisko.OUT.ZadneDverePrave_ZAMKNI THEN
		P3_Pracovisko.STAV.ZadneDvereZamknute:= TRUE;
	ELSE
		P3_Pracovisko.STAV.ZadneDvereZamknute:= FALSE;
	END_IF

	//Stav predné dvere zamknuté//
	IF P3_Pracovisko.OUT.PredneDvereLave_ZAMKNI AND P3_Pracovisko.OUT.PredneDverePrave_ZAMKNI THEN
		P3_Pracovisko.STAV.PredneDvereZamknute:= TRUE;
	ELSE
		P3_Pracovisko.STAV.PredneDvereZamknute:= FALSE;
	END_IF

	//*****************************Reset zóny HV test*****************************************//
	IF Safety.STAV.Linka_ZonaCS_AKTIVNA AND
		(Safety.STAV.P3_Bunka_Zamky_AKTIVNE OR Safety.STAV.P3_VyblokovanieZamkov_AKTIVNE) AND
		NOT Safety.STAV.P3_ZonaHVtest_AKTIVNA AND
		(Safety.STAV.P3_Bunka_VstupBariera_AKTIVNA OR Safety.STAV.P2_Bunka_Zamky_AKTIVNE)AND
		(Safety.STAV.P4_Bunka_VstupBariera_AKTIVNA OR Safety.STAV.P4_Bunka_Zamky_AKTIVNE)THEN
		Safety.OUT.P3_ResetZonyHVtest:= TRUE;
	ELSE
		Safety.OUT.P3_ResetZonyHVtest:= FALSE;
	END_IF

	//*****************************************Reset zóny bunky************************************************//
	IF Safety.STAV.Linka_ZonaCS_AKTIVNA AND
		(Safety.STAV.P3_Bunka_Zamky_AKTIVNE OR Safety.STAV.P3_VyblokovanieZamkov_AKTIVNE) AND
		NOT Safety.STAV.P3_ZonaBunky_AKTIVNA AND
		(Safety.STAV.P3_Bunka_VstupBariera_AKTIVNA OR Safety.STAV.P2_Bunka_Zamky_AKTIVNE)AND
		(Safety.STAV.P4_Bunka_VstupBariera_AKTIVNA OR Safety.STAV.P4_Bunka_Zamky_AKTIVNE)THEN
		Safety.OUT.P3_ResetZonyBunky:= TRUE;
	ELSE
		Safety.OUT.P3_ResetZonyBunky:= FALSE;
	END_IF

END_PROGRAM

PROGRAM _EXIT
	(* Insert code here *)

END_PROGRAM
```

### Program Logical/Program/Pracovisko_4/P4_Main (IEC)

#### Main.st - Init, cyclic, exit code
```iecst
PROGRAM _INIT
	(* Insert code here *)

END_PROGRAM

PROGRAM _CYCLIC

	//Volanie podprogramu//
	ProfinetKomunikaciaKAM14;
	ProfinetKomunikaciaKAM15;
	ProfinetKomunikaciaKAM16;

	//Odomknutie pneumatického zámku zdvižiek//
	IF Safety.STAV.P4_ZonaBunky_AKTIVNA THEN
		P4_Pracovisko.OUT.ZdvizkyPneuZamok_ODOMKNI:= TRUE;
	ELSE
		P4_Pracovisko.OUT.ZdvizkyPneuZamok_ODOMKNI:= FALSE;
	END_IF

	//**************************************Ukončenie cyklu pracoviska****************************************************//
	IF P4_Pracovisko.KoniecCyklu THEN
		IF P4_Dopravniky.Automat THEN
			P4_Dopravniky.KoniecCyklu:= TRUE;
		END_IF
		IF P4_SpodnyStoper.Automat THEN
			P4_SpodnyStoper.KoniecCyklu:= TRUE;
		END_IF
		IF P4_FunkcnyTestA.Automat THEN
			P4_FunkcnyTestA.KoniecCyklu:= TRUE;
		END_IF
		IF P4_FunkcnyTestB.Automat THEN
			P4_FunkcnyTestB.KoniecCyklu:= TRUE;
		END_IF
		IF P4_ZdvizkaZaFunkcTestA.Automat THEN
			P4_ZdvizkaZaFunkcTestA.KoniecCyklu:= TRUE;
		END_IF
		IF P4_ZdvizkaZaFunkcTestB.Automat THEN
			P4_ZdvizkaZaFunkcTestB.KoniecCyklu:= TRUE;
		END_IF
		IF P4_Etiketovacka.Automat THEN
			P4_Etiketovacka.KoniecCyklu:= TRUE;
		END_IF
		IF P4_Vytah.Automat THEN
			P4_Vytah.KoniecCyklu:= TRUE;
		END_IF
		P4_Pracovisko.KoniecCyklu:= FALSE;
	END_IF

	//************************************Ukončenie cyklu pri poruche*****************************************//
	//ST1 - Final test A//
	IF P4_Pracovisko.STAV.Porucha_ST1 THEN
		IF P4_FunkcnyTestA.Automat THEN
			P4_FunkcnyTestA.Reset:= TRUE;
		END_IF
		IF P4_Dopravniky.Automat THEN
			P4_Dopravniky.KoniecCyklu:= TRUE;
		END_IF
		IF P4_SpodnyStoper.Automat THEN
			P4_SpodnyStoper.KoniecCyklu:= TRUE;
		END_IF
		IF P4_FunkcnyTestB.Automat THEN
			P4_FunkcnyTestB.KoniecCyklu:= TRUE;
		END_IF
		IF P4_ZdvizkaZaFunkcTestA.Automat THEN
			P4_ZdvizkaZaFunkcTestA.KoniecCyklu:= TRUE;
		END_IF
		IF P4_ZdvizkaZaFunkcTestB.Automat THEN
			P4_ZdvizkaZaFunkcTestB.KoniecCyklu:= TRUE;
		END_IF
		IF P4_Etiketovacka.Automat THEN
			P4_Etiketovacka.KoniecCyklu:= TRUE;
		END_IF
	END_IF

	//ST2 - Final test B//
	IF P4_Pracovisko.STAV.Porucha_ST2 THEN
		IF P4_FunkcnyTestB.Automat THEN
			P4_FunkcnyTestB.Reset:= TRUE;
		END_IF
		IF P4_Dopravniky.Automat THEN
			P4_Dopravniky.KoniecCyklu:= TRUE;
		END_IF
		IF P4_SpodnyStoper.Automat THEN
			P4_SpodnyStoper.KoniecCyklu:= TRUE;
		END_IF
		IF P4_FunkcnyTestA.Automat THEN
			P4_FunkcnyTestA.KoniecCyklu:= TRUE;
		END_IF
		IF P4_ZdvizkaZaFunkcTestA.Automat THEN
			P4_ZdvizkaZaFunkcTestA.KoniecCyklu:= TRUE;
		END_IF
		IF P4_ZdvizkaZaFunkcTestB.Automat THEN
			P4_ZdvizkaZaFunkcTestB.KoniecCyklu:= TRUE;
		END_IF
		IF P4_Etiketovacka.Automat THEN
			P4_Etiketovacka.KoniecCyklu:= TRUE;
		END_IF
	END_IF

	//ST3 - Zdvižka za final testom A//
	IF P4_Pracovisko.STAV.Porucha_ST3 THEN
		IF P4_ZdvizkaZaFunkcTestA.Automat THEN
			P4_ZdvizkaZaFunkcTestA.Reset:= TRUE;
		END_IF
		IF P4_Dopravniky.Automat THEN
			P4_Dopravniky.KoniecCyklu:= TRUE;
		END_IF
		IF P4_SpodnyStoper.Automat THEN
			P4_SpodnyStoper.KoniecCyklu:= TRUE;
		END_IF
		IF P4_FunkcnyTestA.Automat THEN
			P4_FunkcnyTestA.KoniecCyklu:= TRUE;
		END_IF
		IF P4_FunkcnyTestB.Automat THEN
			P4_FunkcnyTestB.KoniecCyklu:= TRUE;
		END_IF
		IF P4_ZdvizkaZaFunkcTestB.Automat THEN
			P4_ZdvizkaZaFunkcTestB.KoniecCyklu:= TRUE;
		END_IF
		IF P4_Etiketovacka.Automat THEN
			P4_Etiketovacka.KoniecCyklu:= TRUE;
		END_IF
	END_IF

	//ST4 - Zdvižka za final testom B//
	IF P4_Pracovisko.STAV.Porucha_ST4 THEN
		IF P4_ZdvizkaZaFunkcTestB.Automat THEN
			P4_ZdvizkaZaFunkcTestB.Reset:= TRUE;
		END_IF
		IF P4_Dopravniky.Automat THEN
			P4_Dopravniky.KoniecCyklu:= TRUE;
		END_IF
		IF P4_SpodnyStoper.Automat THEN
			P4_SpodnyStoper.KoniecCyklu:= TRUE;
		END_IF
		IF P4_FunkcnyTestA.Automat THEN
			P4_FunkcnyTestA.KoniecCyklu:= TRUE;
		END_IF
		IF P4_FunkcnyTestB.Automat THEN
			P4_FunkcnyTestB.KoniecCyklu:= TRUE;
		END_IF
		IF P4_ZdvizkaZaFunkcTestA.Automat THEN
			P4_ZdvizkaZaFunkcTestA.KoniecCyklu:= TRUE;
		END_IF
		IF P4_Etiketovacka.Automat THEN
			P4_Etiketovacka.KoniecCyklu:= TRUE;
		END_IF
	END_IF

	//ST5 - Etiketovanie//
	IF P4_Pracovisko.STAV.Porucha_ST5 THEN
		IF P4_Dopravniky.Automat THEN
			P4_Dopravniky.KoniecCyklu:= TRUE;
		END_IF
		IF P4_SpodnyStoper.Automat THEN
			P4_SpodnyStoper.KoniecCyklu:= TRUE;
		END_IF
		IF P4_FunkcnyTestA.Automat THEN
			P4_FunkcnyTestA.KoniecCyklu:= TRUE;
		END_IF
		IF P4_FunkcnyTestB.Automat THEN
			P4_FunkcnyTestB.KoniecCyklu:= TRUE;
		END_IF
		IF P4_ZdvizkaZaFunkcTestA.Automat THEN
			P4_ZdvizkaZaFunkcTestA.KoniecCyklu:= TRUE;
		END_IF
		IF P4_ZdvizkaZaFunkcTestB.Automat THEN
			P4_ZdvizkaZaFunkcTestB.KoniecCyklu:= TRUE;
		END_IF
	END_IF

	//ST6 - Výťah//
	IF P4_Pracovisko.STAV.Porucha_ST6 THEN
		IF P4_Vytah.Automat THEN
			P4_Vytah.Reset:= TRUE;
		END_IF
	END_IF

	//*********************************Status prebieha ukončenie cyklu********************************************//
	IF P4_Dopravniky.KoniecCyklu OR
		P4_SpodnyStoper.KoniecCyklu OR
		P4_FunkcnyTestA.KoniecCyklu OR
		P4_FunkcnyTestB.KoniecCyklu OR
		P4_ZdvizkaZaFunkcTestA.KoniecCyklu OR
		P4_ZdvizkaZaFunkcTestB.KoniecCyklu OR
		P4_Etiketovacka.KoniecCyklu OR
		P4_Vytah.KoniecCyklu THEN
		P4_Pracovisko.STAV.UkoncenieCyklu_BUSY:= TRUE;
	ELSE
		P4_Pracovisko.STAV.UkoncenieCyklu_BUSY:= FALSE;
	END_IF

	//*******************************Resetovanie pracoviska po stlačení tlačítka Automat******************************************//
	IF P34_Vizu.TL_RezimAutomat THEN
		IF P3_Pracovisko.STAV.Manual THEN
			P3_Pracovisko.Reset:= TRUE;
		END_IF
		IF P4_Pracovisko.STAV.Manual THEN
			P4_Pracovisko.Reset:= TRUE;
		END_IF
		P34_Vizu.TL_RezimAutomat:= FALSE;
	END_IF

	//******************************************Resetovanie pracoviska************************************************************//
	IF P4_Pracovisko.Reset THEN
		P4_Dopravniky.Reset:= TRUE;
		P4_SpodnyStoper.Reset:= TRUE;
		P4_FunkcnyTestA.Reset:= TRUE;
		P4_FunkcnyTestB.Reset:= TRUE;
		P4_ZdvizkaZaFunkcTestA.Reset:= TRUE;
		P4_ZdvizkaZaFunkcTestB.Reset:= TRUE;
		P4_Etiketovacka.Reset:= TRUE;
		P4_Vytah.Reset:= TRUE;
		P4_Pracovisko.STAV.Porucha_ST1:= FALSE;
		P4_Pracovisko.STAV.Porucha_ST2:= FALSE;
		P4_Pracovisko.STAV.Porucha_ST3:= FALSE;
		P4_Pracovisko.STAV.Porucha_ST4:= FALSE;
		P4_Pracovisko.STAV.Porucha_ST5:= FALSE;
		P4_Pracovisko.STAV.Porucha_ST6:= FALSE;
		P4_Pracovisko.Reset:= FALSE;
	END_IF

	//Prepnutie pracoviska do manualneho režimu//
	IF P4_Pracovisko.Manual THEN
		P4_Dopravniky.Manual:= TRUE;
		P4_SpodnyStoper.Manual:= TRUE;
		P4_FunkcnyTestA.Manual:= TRUE;
		P4_FunkcnyTestB.Manual:= TRUE;
		P4_ZdvizkaZaFunkcTestA.Manual:= TRUE;
		P4_ZdvizkaZaFunkcTestB.Manual:= TRUE;
		P4_Etiketovacka.Manual:= TRUE;
		P4_Vytah.Manual:= TRUE;
		P4_Pracovisko.Manual:= FALSE;
	END_IF

	//Spustenie pracoviska v automatickom režime//
	IF P4_Pracovisko.Automat THEN
		IF Safety.STAV.P4_ZonaVytahu_AKTIVNA AND P4_Pracovisko.STAV.HardwareVytahu_OK THEN
			P4_Vytah.Automat:= TRUE;
		END_IF
		IF Safety.STAV.P4_ZonaBunky_AKTIVNA AND P4_Pracovisko.STAV.HardwareBunky_OK THEN
			P4_Dopravniky.Automat:= TRUE;
			P4_SpodnyStoper.Automat:= TRUE;
			P4_FunkcnyTestA.Automat:= TRUE;
			P4_FunkcnyTestB.Automat:= TRUE;
			P4_ZdvizkaZaFunkcTestA.Automat:= TRUE;
			P4_ZdvizkaZaFunkcTestB.Automat:= TRUE;
			P4_Etiketovacka.Automat:= TRUE;
		END_IF
		P4_Pracovisko.Automat:= FALSE;
	END_IF

	//***************************************************Príznaky pracoviska******************************************************//
	//Príznak pracovisko stav AUTOMAT//
	IF P4_Dopravniky.Automat OR
		P4_SpodnyStoper.Automat OR
		P4_FunkcnyTestA.Automat OR
		P4_FunkcnyTestB.Automat OR
		P4_ZdvizkaZaFunkcTestA.Automat OR
		P4_ZdvizkaZaFunkcTestB.Automat OR
		P4_Etiketovacka.Automat OR
		P4_Vytah.Automat THEN
		P4_Pracovisko.STAV.Automat:= TRUE;
	ELSE
		P4_Pracovisko.STAV.Automat:= FALSE;
	END_IF

	//Priznak pracovisko stav MANUAL//
	IF P4_Dopravniky.Manual OR
		P4_SpodnyStoper.Manual OR
		P4_FunkcnyTestA.Manual OR
		P4_FunkcnyTestB.Manual OR
		P4_ZdvizkaZaFunkcTestA.Manual OR
		P4_ZdvizkaZaFunkcTestB.Manual OR
		P4_Etiketovacka.Manual OR
		P4_Vytah.Manual THEN
		P4_Pracovisko.STAV.Manual:= TRUE;
	ELSE
		P4_Pracovisko.STAV.Manual:= FALSE;
	END_IF

	//Príznak pracovisko stav PoINIT//
	IF P4_Dopravniky.STAV.PoINIT AND
		P4_SpodnyStoper.STAV.PoINIT AND
		P4_FunkcnyTestA.STAV.PoINIT AND
		P4_FunkcnyTestB.STAV.PoINIT AND
		P4_ZdvizkaZaFunkcTestA.STAV.PoINIT AND
		P4_ZdvizkaZaFunkcTestB.STAV.PoINIT AND
		P4_Etiketovacka.STAV.PoINIT AND
		P4_Vytah.STAV.PoINIT THEN
		P4_Pracovisko.STAV.PoINIT:= TRUE;
	ELSE
		P4_Pracovisko.STAV.PoINIT:= FALSE;
	END_IF

	//Príznak pracovisko stav READY//
	IF SC_P4_Dopravniky.Step = 1 AND
		SC_P4_SpodnyStoper.Step = 1 AND
		SC_P4_FunkcnyTestA.Step = 1 AND
		SC_P4_FunkcnyTestB.Step = 1 AND
		SC_P4_ZdvizkaZaFunkcTestA.Step = 1 AND
		SC_P4_ZdvizkaZaFunkcTestB.Step = 1 AND
		SC_P4_Etiketovacka.Step = 1 AND
		SC_P4_Vytah.Step = 1 THEN
		P4_Pracovisko.STAV.READY:= TRUE;
	ELSE
		P4_Pracovisko.STAV.READY:= FALSE;
	END_IF

	//Príznak pracovisko stav PORUCHA//
	IF P4_Pracovisko.STAV.Porucha_ST1 OR
		P4_Pracovisko.STAV.Porucha_ST2 OR
		P4_Pracovisko.STAV.Porucha_ST3 OR
		P4_Pracovisko.STAV.Porucha_ST4 OR
		P4_Pracovisko.STAV.Porucha_ST5 OR
		P4_Pracovisko.STAV.Porucha_ST6 THEN
		P4_Pracovisko.STAV.PORUCHA:= TRUE;
	ELSE
		P4_Pracovisko.STAV.PORUCHA:= FALSE;
	END_IF

	//Priznak HW Vytahu OK//
	IF P4_Pracovisko.IN.TlakVzduchu_OK AND
		P4_Pracovisko.IN.ModulFesto_IO_KomOK AND
		P4_Pracovisko.IN.ModulWeidmuller_IO_KomOK AND
		P4_Pracovisko.IN.ServoZdvihuVytahu_KomOK AND
		P3_Pracovisko.IN.Kamery_ControlUnit_KomOK AND
		P4_Pracovisko.IN.VentilovyTerminal_KomOK THEN
		P4_Pracovisko.STAV.HardwareVytahu_OK:= TRUE;
	ELSE
		P4_Pracovisko.STAV.HardwareVytahu_OK:= FALSE;
	END_IF

	//Príznak HW Bunky OK//
	IF P4_Pracovisko.IN.TlakVzduchu_OK AND
		P4_Pracovisko.IN.ModulFesto_IO_KomOK AND
		P4_Pracovisko.IN.ModulWeidmuller_IO_KomOK AND
		P4_Pracovisko.IN.ServoZdvihuAplikEtikiet_KomOK AND
		P4_Pracovisko.IN.SmartKamera14_KomOK AND
		P3_Pracovisko.IN.Kamery_ControlUnit_KomOK AND
		P4_Pracovisko.IN.VentilovyTerminal_KomOK THEN
		P4_Pracovisko.STAV.HardwareBunky_OK:= TRUE;
	ELSE
		P4_Pracovisko.STAV.HardwareBunky_OK:= FALSE;
	END_IF

	//Priznak Funkčný Test A zasunuty//
	IF P4_FunkcnyTestA.IN.Centrovanie_ZASUNUTE AND P4_FunkcnyTestA.IN.HorneKontakty_ZASUNUTE AND P4_FunkcnyTestA.IN.SpodneKontakty_ZASUNUTE THEN
		P4_Pracovisko.STAV.FunkcnyTestA_Zasunuty:= TRUE;
	ELSE
		P4_Pracovisko.STAV.FunkcnyTestA_Zasunuty:= FALSE;
	END_IF

	//Priznak Funkčný Test B zasunuty//
	IF P4_FunkcnyTestB.IN.Centrovanie_ZASUNUTE AND P4_FunkcnyTestB.IN.HorneKontakty_ZASUNUTE AND P4_FunkcnyTestB.IN.SpodneKontakty_ZASUNUTE THEN
		P4_Pracovisko.STAV.FunkcnyTestB_Zasunuty:= TRUE;
	ELSE
		P4_Pracovisko.STAV.FunkcnyTestB_Zasunuty:= FALSE;
	END_IF

	//*****************************Zapnutie osvetlenia pracoviska*********************************************************//
	P4_Pracovisko.OUT.OsvetlenieBunky_ON:= FALSE;
	P4_Vytah.OUT.OsvetlenieVytahu_ON:= TRUE;
	P4_Pracovisko.OUT.Osvetlenie_CAM15_ON:= TRUE;
	//****************************************Ovládanie majáka***********************************************//
	//Zelené svetlo//

	IF P4_Pracovisko.STAV.Automat THEN
		P4_Pracovisko.OUT.Majak_ZeleneSvetlo_ON:= TRUE;
	ELSIF P4_Pracovisko.STAV.Manual THEN
		P4_Pracovisko.OUT.Majak_ZeleneSvetlo_ON:= Blikac500ms;
	ELSE
		P4_Pracovisko.OUT.Majak_ZeleneSvetlo_ON:= FALSE;
	END_IF

	//Oranžové svetlo//
	IF P4_Pracovisko.STAV.Automat AND NOT P4_Pracovisko.STAV.PoINIT THEN
		P4_Pracovisko.OUT.Majak_OranzoveSvetlo_ON:= TRUE;
	ELSE
		P4_Pracovisko.OUT.Majak_OranzoveSvetlo_ON:= FALSE;
	END_IF

	//Červené svetlo//
	IF NOT Safety.STAV.Linka_ZonaCS_AKTIVNA THEN
		P4_Pracovisko.OUT.Majak_CerveneSvetlo_ON:= TRUE;
	ELSIF P4_Pracovisko.STAV.Porucha_ST1 THEN
		P4_Pracovisko.OUT.Majak_CerveneSvetlo_ON:= TRUE;
	ELSIF P4_Pracovisko.STAV.Porucha_ST2 THEN
		P4_Pracovisko.OUT.Majak_CerveneSvetlo_ON:= TRUE;
	ELSIF P4_Pracovisko.STAV.Porucha_ST3 THEN
		P4_Pracovisko.OUT.Majak_CerveneSvetlo_ON:= TRUE;
	ELSIF P4_Pracovisko.STAV.Porucha_ST4 THEN
		P4_Pracovisko.OUT.Majak_CerveneSvetlo_ON:= TRUE;
	ELSIF P4_Pracovisko.STAV.Porucha_ST5 THEN
		P4_Pracovisko.OUT.Majak_CerveneSvetlo_ON:= TRUE;
	ELSIF P4_Pracovisko.STAV.Porucha_ST6 THEN
		P4_Pracovisko.OUT.Majak_CerveneSvetlo_ON:= TRUE;
	ELSE
		P4_Pracovisko.OUT.Majak_CerveneSvetlo_ON:= FALSE;
	END_IF

	//Zvuková signalizácia//
//	IF EDGEPOS(P4_Pracovisko.STAV.Porucha_ST1) THEN
//		P4_Pracovisko.OUT.Majak_Hukacka_ON:= Blikac500ms;
//	ELSIF EDGEPOS(P4_Pracovisko.STAV.Porucha_ST2) THEN
//		P4_Pracovisko.OUT.Majak_Hukacka_ON:= Blikac500ms;
//	ELSIF EDGEPOS(P4_Pracovisko.STAV.Porucha_ST3) THEN
//		P4_Pracovisko.OUT.Majak_Hukacka_ON:= Blikac500ms;
//	ELSIF EDGEPOS(P4_Pracovisko.STAV.Porucha_ST4) THEN
//		P4_Pracovisko.OUT.Majak_Hukacka_ON:= Blikac500ms;
//	ELSIF EDGEPOS(P4_Pracovisko.STAV.Porucha_ST5) THEN
//		P4_Pracovisko.OUT.Majak_Hukacka_ON:= Blikac500ms;
//	ELSIF EDGEPOS(P4_Pracovisko.STAV.Porucha_ST6) THEN
//		P4_Pracovisko.OUT.Majak_Hukacka_ON:= Blikac500ms;
//	END_IF

END_PROGRAM

PROGRAM _EXIT
	(* Insert code here *)

END_PROGRAM
```

#### Variables.var - Local variables
```iecst
VAR
	Convert_0 : UsintToUint := (0);
	Convert_1 : UsintToUint := (0);
	Convert_2 : UsintToUint := (0);
END_VAR
```

#### ProfinetKomunikaciaKAM14.st
```iecst
ACTION ProfinetKomunikaciaKAM14:
	//Smart kamera//

	CAM14.STAV.READY:= P4_Pracovisko.IN.SmartKamera14_KomOK;

	//Vstupy pre kameru//
	CAM14.Profinet_PLC_OUTPUTS[0].0:= CAM14.CMD.Triger;

	//Výstupy z kamery//
	CAM14.STAV.SWITCH:= CAM14.Profinet_PLC_INPUTS[12].0;

	//Výsledky kamery//
	CAM14.RESULT.PowerCP.CitanieQRkodu_PowerCP_OK:= CAM14.Profinet_PLC_INPUTS[0].0;

	//Prečítaný QR kód DPS//
	IF EDGE(CAM14.STAV.SWITCH) THEN
		brsstrcpy(ADR(CAM14.RESULT.PowerCP.PrecitanyQRkod_PowerCP),ADR(CAM14.Profinet_QRkod_Znaky));
	END_IF

	//Stav výsledky READY//
	IF EDGE(CAM14.STAV.SWITCH)THEN
		CAM14.STAV.Results_READY:= TRUE;
	END_IF

	//Run counter kamery//
	Convert_0.IN_Byte0:= CAM14.STAV.RunCounter_Byte1;
	Convert_0.IN_Byte1:= CAM14.STAV.RunCounter_Byte0;

	CAM14.STAV.RunCounter:= Convert_0.OUT_UINT;
	Convert_0();

END_ACTION
```

#### ProfinetKomunikaciaKAM15.st
```iecst
ACTION ProfinetKomunikaciaKAM15:
	//Control Unit CAM 10//

	//Vstupy pre kameru//
	CAM15.Profinet_PLC_OUTPUTS[0].3:= CAM15.CMD.Triger;

	//Výstupy z kamery//
	CAM15.STAV.READY:= CAM15.Profinet_PLC_INPUTS[0].0;
	CAM15.STAV.SWITCH:= CAM15.Profinet_PLC_INPUTS[0].1;
    CAM15.STAV.BUSY:= CAM15.Profinet_PLC_INPUTS[0].2;
    CAM15.STAV.Command_AKCEPTOVANY:= CAM15.Profinet_PLC_INPUTS[0].3;
    CAM15.STAV.Command_READY:= CAM15.Profinet_PLC_INPUTS[0].4;
    CAM15.STAV.Command_ERROR:= CAM15.Profinet_PLC_INPUTS[0].5;

	//Výsledky kamery//

	//Výsledky kamery//
	CAM15.RESULT.Pritomn_Etikety:= CAM15.Profinet_PLC_INPUTS[2].0;
	CAM15.RESULT.Pritomn_LogoBMV:= CAM15.Profinet_PLC_INPUTS[2].1;
	CAM15.RESULT.Pritomn_LogoPanasonic:= CAM15.Profinet_PLC_INPUTS[2].2;
	CAM15.RESULT.CitanieQRkodu_Etikety_OK:= CAM15.Profinet_PLC_INPUTS[2].3;

	//Stav výsledky READY//
	IF EDGE(CAM15.STAV.SWITCH)THEN
		CAM15.STAV.Results_READY:= TRUE;
		brsstrcpy(ADR(CAM15.RESULT.PrecitanyQRkod_Etikety),ADR(CAM15.Profinet_QRkod_Znaky));
		CAM15_PocetFotiek:= CAM15_PocetFotiek + 1;
	END_IF

	//Vymazanie adresára kamery//
	IF EDGEPOS(CAM15_PocetFotiek > 50) THEN
		FTP_CAM15.CMD.VymazFotku:= TRUE;
		FTP_CAM15.STATUS.VymazanieAdresaraKamery_BUSY:= TRUE;
	END_IF

	IF (FTP_CAM15.STATUS.KomunikaciaUkoncena OR FTP_CAM15.STATUS.KomunikaciaError) AND FTP_CAM15.STATUS.VymazanieAdresaraKamery_BUSY THEN
		FTP_CAM15.CMD.VymazFotku:= FALSE;
		FTP_CAM15.STATUS.VymazanieAdresaraKamery_BUSY:= FALSE;
	END_IF

	//Run counter kamery//
	Convert_1.IN_Byte0:= CAM15.STAV.RunCounter_Byte1;
	Convert_1.IN_Byte1:= CAM15.STAV.RunCounter_Byte0;

	CAM15.STAV.RunCounter:= Convert_1.OUT_UINT;
	Convert_1();

END_ACTION
```

#### ProfinetKomunikaciaKAM16.st
```iecst
ACTION ProfinetKomunikaciaKAM16:
	//Control Unit CAM 11//

	//Vstupy pre kameru//
	CAM16.Profinet_PLC_OUTPUTS[0].3:= CAM16.CMD.Triger;

	//Výstupy z kamery//
	CAM16.STAV.READY:= CAM16.Profinet_PLC_INPUTS[0].0;
	CAM16.STAV.SWITCH:= CAM16.Profinet_PLC_INPUTS[0].1;
    CAM16.STAV.BUSY:= CAM16.Profinet_PLC_INPUTS[0].2;
    CAM16.STAV.Command_AKCEPTOVANY:= CAM16.Profinet_PLC_INPUTS[0].3;
    CAM16.STAV.Command_READY:= CAM16.Profinet_PLC_INPUTS[0].4;
    CAM16.STAV.Command_ERROR:= CAM16.Profinet_PLC_INPUTS[0].5;

	//Výsledky kamery//
	CAM16.RESULT.Paletka.Pritomn_PowerCP:= CAM16.Profinet_PLC_INPUTS[2].0;
	CAM16.RESULT.Paletka.Pritomn_Busbarov_4F:= CAM16.Profinet_PLC_INPUTS[2].1;
	CAM16.RESULT.Paletka.Pritomn_Busbarov_5F:= CAM16.Profinet_PLC_INPUTS[2].2;
	CAM16.RESULT.Paletka.Pritomn_Busbarov_5H:= CAM16.Profinet_PLC_INPUTS[2].3;
	CAM16.RESULT.Paletka.Pritomn_LavyMVcase:= CAM16.Profinet_PLC_INPUTS[2].4;
    CAM16.RESULT.Paletka.Pritomn_PravyMVcase:= CAM16.Profinet_PLC_INPUTS[2].5;

	//Stav výsledky READY//
	IF EDGE(CAM16.STAV.SWITCH)THEN
		CAM16.STAV.Results_READY:= TRUE;
		CAM16_PocetFotiek:= CAM16_PocetFotiek + 1;
	END_IF

	//Vymazanie adresára kamery//
	IF EDGEPOS(CAM16_PocetFotiek > 50) THEN
		FTP_CAM16.CMD.VymazFotku:= TRUE;
		FTP_CAM16.STATUS.VymazanieAdresaraKamery_BUSY:= TRUE;
	END_IF

	IF (FTP_CAM16.STATUS.KomunikaciaUkoncena OR FTP_CAM16.STATUS.KomunikaciaError) AND FTP_CAM16.STATUS.VymazanieAdresaraKamery_BUSY THEN
		FTP_CAM16.CMD.VymazFotku:= FALSE;
		FTP_CAM16.STATUS.VymazanieAdresaraKamery_BUSY:= FALSE;
	END_IF

	//Run counter kamery//
	Convert_2.IN_Byte0:= CAM16.STAV.RunCounter_Byte1;
	Convert_2.IN_Byte1:= CAM16.STAV.RunCounter_Byte0;

	CAM16.STAV.RunCounter:= Convert_2.OUT_UINT;
	Convert_2();

END_ACTION
```

### Program Logical/Program/Pracovisko_4/P4_Dopravniky (IEC)

#### Main.st - Init, cyclic, exit code
```iecst
PROGRAM _INIT
	(* Insert code here *)

END_PROGRAM

PROGRAM _CYCLIC

	//Volanie funkcie SequenceControl//
	SequenceControl(SC:= SC_P4_Dopravniky);

	//Reset sekcie //
	IF P4_Dopravniky.Reset THEN
		SC_P4_Dopravniky.Step:= 0;
		P4_Dopravniky.Reset:= FALSE;
	ELSIF NOT Safety.STAV.Linka_ZonaCS_AKTIVNA THEN
		SC_P4_Dopravniky.Step:= 0;
	END_IF

	CASE SC_P4_Dopravniky.Step OF

		0:
			SC_P4_Dopravniky.StepName:='0 - Nulovanie';
			P4_Dopravniky.Automat:= FALSE;
			P4_Dopravniky.KoniecCyklu:= FALSE;
			P4_Dopravniky.Manual:= FALSE;
			P4_Dopravniky.STAV.PoINIT:= FALSE;
			P4_Dopravniky.OUT.PrednyDopravnikBunky_ON:= FALSE;
			P4_Dopravniky.OUT.PriecnyDopravnik_VPRED:= FALSE;
			P4_Dopravniky.OUT.VratnyDopravnik_ON:= FALSE;
			P4_Dopravniky.OUT.ZadnyDopravnikBunky_ON:= FALSE;

			IF Safety.STAV.Linka_ZonaCS_AKTIVNA AND
				Safety.STAV.P4_ZonaBunky_AKTIVNA AND
				P4_Pracovisko.STAV.HardwareBunky_OK AND
				NOT P4_Pracovisko.STAV.Porucha_ST1 AND
				NOT P4_Pracovisko.STAV.Porucha_ST2 AND
				NOT P4_Pracovisko.STAV.Porucha_ST3 AND
				NOT P4_Pracovisko.STAV.Porucha_ST4 AND
				NOT P4_Pracovisko.STAV.Porucha_ST5 AND
				NOT P4_Pracovisko.STAV.Porucha_ST6 THEN
				SC_P4_Dopravniky.ResetStep:= TRUE;
				SC_P4_Dopravniky.Step:= 1;
			END_IF

		1:
			SC_P4_Dopravniky.StepName:='1 - Cakam na spustenie vyroby';
			P4_Dopravniky.KoniecCyklu:= FALSE;
			IF P4_Dopravniky.Automat THEN
				SC_P4_Dopravniky.Step:= 2;
			ELSIF P4_Dopravniky.Manual THEN
				SC_P4_Dopravniky.Step:= 700;
			END_IF

			//********************************************************Inicializácia****************************************************************************//

		2:
			SC_P4_Dopravniky.StepName:='2 - Inicializacia - cakam na spustenie inicializacie';
			SC_P4_Dopravniky.IdleTime.PT:= T#1s;
			SC_P4_Dopravniky.AlarmTime.PT:= T#5s;

			IF P4_Pracovisko.STAV.FunkcnyTestA_Zasunuty AND P4_Pracovisko.STAV.FunkcnyTestB_Zasunuty THEN
				SC_P4_Dopravniky.IdleTime.IN:= TRUE;
			ELSE
				SC_P4_Dopravniky.IdleTime.IN:= FALSE;
			END_IF

			IF SC_P4_Dopravniky.IdleTime.Q THEN
				SC_P4_Dopravniky.ResetStep:= TRUE;
				SC_P4_Dopravniky.Step:= 3;
			END_IF

		3:
			SC_P4_Dopravniky.StepName:='3 - Inicializacia - inicializacia tlmenia stoprov';
			SC_P4_Dopravniky.IdleTime.PT:= T#1s;
			SC_P4_Dopravniky.AlarmTime.PT:= T#5s;

			IF P4_FunkcnyTestA.RFID_hlava.PritomnostPaletky AND
				P4_FunkcnyTestB.RFID_hlava.PritomnostPaletky AND
				P4_ZdvizkaZaFunkcTestA.IN.PritomnostPaletky AND
				P4_ZdvizkaZaFunkcTestB.IN.PritomnostPaletky AND
				P4_SpodnyStoper.IN.PritomnostPaletky AND
				P4_Etiketovacka.RFID_hlava.PritomnostPaletky THEN
				SC_P4_Dopravniky.ResetStep:= TRUE;
				SC_P4_Dopravniky.Step:= 5;
			ELSE
				IF NOT P4_FunkcnyTestA.RFID_hlava.PritomnostPaletky AND P4_FunkcnyTestA.IN.Centrovanie_ZASUNUTE THEN
					P4_FunkcnyTestA.OUT.ZasunStoper:= TRUE;
				END_IF
				IF NOT P4_FunkcnyTestB.RFID_hlava.PritomnostPaletky AND P4_FunkcnyTestB.IN.Centrovanie_ZASUNUTE THEN
					P4_FunkcnyTestB.OUT.ZasunStoper:= TRUE;
				END_IF
				IF NOT P4_SpodnyStoper.IN.PritomnostPaletky THEN
					P4_SpodnyStoper.OUT.ZasunStoper:= TRUE;
				END_IF
				IF NOT P4_ZdvizkaZaFunkcTestA.IN.PritomnostPaletky AND P4_ZdvizkaZaFunkcTestA.IN.Zdvizka_StrednaPoloha THEN
					P4_ZdvizkaZaFunkcTestA.OUT.TlmicPaletky_ZASUN:= FALSE;
					P4_ZdvizkaZaFunkcTestA.OUT.TlmicPaletky_VYSUN:= TRUE;
				END_IF
				IF NOT P4_ZdvizkaZaFunkcTestB.IN.PritomnostPaletky AND P4_ZdvizkaZaFunkcTestB.IN.Zdvizka_StrednaPoloha THEN
					P4_ZdvizkaZaFunkcTestB.OUT.TlmicPaletky_VYSUN:= TRUE;
				END_IF
				IF NOT P4_Etiketovacka.RFID_hlava.PritomnostPaletky AND P4_Etiketovacka.IN.Centrovanie_ZASUNUTE THEN
					P4_Etiketovacka.OUT.ZasunStoper:= TRUE;
				END_IF
				SC_P4_Dopravniky.IdleTime.IN:= TRUE;
			END_IF

			IF SC_P4_Dopravniky.IdleTime.Q THEN
				P4_FunkcnyTestA.OUT.ZasunStoper:= FALSE;
				P4_FunkcnyTestB.OUT.ZasunStoper:= FALSE;
				P4_SpodnyStoper.OUT.ZasunStoper:= FALSE;
				P4_ZdvizkaZaFunkcTestA.OUT.TlmicPaletky_ZASUN:= FALSE;
				P4_ZdvizkaZaFunkcTestA.OUT.TlmicPaletky_VYSUN:= FALSE;
				P4_ZdvizkaZaFunkcTestB.OUT.TlmicPaletky_VYSUN:= FALSE;
				P4_Etiketovacka.OUT.ZasunStoper:= FALSE;
				SC_P4_Dopravniky.ResetStep:= TRUE;
				SC_P4_Dopravniky.Step:= 5;
			END_IF

		5:
			SC_P4_Dopravniky.StepName:='5 - Inicializacia - ukoncenie inicializacie';
			SC_P4_Dopravniky.IdleTime.PT:= T#5s;
			SC_P4_Dopravniky.AlarmTime.PT:= T#5s;

			P4_Dopravniky.OUT.PrednyDopravnikBunky_ON:= TRUE;
			P4_Dopravniky.OUT.ZadnyDopravnikBunky_ON:= TRUE;
			P4_Dopravniky.OUT.VratnyDopravnik_ON:= TRUE;
			SC_P4_Dopravniky.IdleTime.IN:= TRUE;

			IF SC_P4_Dopravniky.IdleTime.Q THEN
				P4_Dopravniky.STAV.PoINIT:= TRUE;
				SC_P4_Dopravniky.ResetStep:= TRUE;
				SC_P4_Dopravniky.Step:= 100;
			END_IF

		//********************************************************Automatický režim****************************************************************************//

		100:
			SC_P4_Dopravniky.StepName:='100 - Automaticky Rezim - cakam na vypnutie dopravnikou';
			SC_P4_Dopravniky.IdleTime.PT:= T#200ms;
			SC_P4_Dopravniky.AlarmTime.PT:= T#5s;

			IF P4_Dopravniky.KoniecCyklu AND
				NOT P4_FunkcnyTestA.Automat AND
				NOT P4_FunkcnyTestB.Automat AND
				NOT P4_ZdvizkaZaFunkcTestA.Automat AND
				NOT P4_ZdvizkaZaFunkcTestB.Automat AND
				NOT P4_Etiketovacka.Automat AND
				NOT P4_SpodnyStoper.Automat AND
				NOT P4_Vytah.Automat THEN
				SC_P4_Dopravniky.ResetStep:= TRUE;
				SC_P4_Dopravniky.Step:= 0;
			END_IF

			//*******************************************************Manuálny režim*******************************************************************************//
		700:
			SC_P4_Dopravniky.StepName:='700 - Manualny Rezim';
			SC_P4_Dopravniky.IdleTime.PT:= T#8s;
			SC_P4_Dopravniky.AlarmTime.PT:= T#5s;

	END_CASE

END_PROGRAM

PROGRAM _EXIT
	(* Insert code here *)

END_PROGRAM
```

### Program Logical/Program/Pracovisko_4/P4_SpodnyStoper (IEC)

#### Main.st - Init, cyclic, exit code
```iecst
PROGRAM _INIT
	(* Insert code here *)

END_PROGRAM

PROGRAM _CYCLIC

	//Volanie funkcie SequenceControl//
	SequenceControl(SC:= SC_P4_SpodnyStoper);

	//Reset sekcie //
	IF P4_SpodnyStoper.Reset THEN
		SC_P4_SpodnyStoper.Step:= 0;
		P4_SpodnyStoper.Reset:= FALSE;
	ELSIF NOT Safety.STAV.Linka_ZonaCS_AKTIVNA THEN
		SC_P4_SpodnyStoper.Step:= 0;
	END_IF

	CASE SC_P4_SpodnyStoper.Step OF

		0:
			SC_P4_SpodnyStoper.StepName:='0 - Nulovanie';
			P4_SpodnyStoper.Automat:= FALSE;
			P4_SpodnyStoper.KoniecCyklu:= FALSE;
			P4_SpodnyStoper.Manual:= FALSE;
			P4_SpodnyStoper.STAV.PoINIT:= FALSE;
			P4_SpodnyStoper.STAV.PrebiehaVyvezeniePaletky:= FALSE;
			P4_SpodnyStoper.OUT.ZasunStoper:= FALSE;

			IF Safety.STAV.Linka_ZonaCS_AKTIVNA AND
				Safety.STAV.P4_ZonaBunky_AKTIVNA AND
				P4_Pracovisko.STAV.HardwareBunky_OK THEN
				SC_P4_SpodnyStoper.ResetStep:= TRUE;
				SC_P4_SpodnyStoper.Step:= 1;
			END_IF

		1:
			SC_P4_SpodnyStoper.StepName:='1 - Cakam na spustenie vyroby';
			P4_SpodnyStoper.KoniecCyklu:= FALSE;
			IF P4_SpodnyStoper.Automat THEN
				SC_P4_SpodnyStoper.Step:= 2;
			ELSIF P4_SpodnyStoper.Manual THEN
				SC_P4_SpodnyStoper.Step:= 700;
			END_IF

			//********************************************************Inicializácia****************************************************************************//
		2:
			SC_P3_SpodnyStoper.StepName:='2 - Inicializacia - cakam na spustenie inicializacie';
			SC_P3_SpodnyStoper.IdleTime.PT:= T#4s;
			SC_P3_SpodnyStoper.AlarmTime.PT:= T#5s;

			IF P4_Dopravniky.STAV.PoINIT THEN
				SC_P4_SpodnyStoper.ResetStep:= TRUE;
				SC_P4_SpodnyStoper.Step:= 3;
			END_IF

		3:
			SC_P4_SpodnyStoper.StepName:='3 - Inicializacia - hladanie paletky';
			SC_P4_SpodnyStoper.IdleTime.PT:= T#5s;
			SC_P4_SpodnyStoper.AlarmTime.PT:= T#5s;
			SC_P4_SpodnyStoper.IdleTime.IN:= TRUE;

			IF P4_SpodnyStoper.IN.PritomnostPaletky THEN
				P4_SpodnyStoper.STAV.PoINIT:= TRUE;
				SC_P4_SpodnyStoper.ResetStep:= TRUE;
				SC_P4_SpodnyStoper.Step:= 101;
			ELSIF SC_P4_SpodnyStoper.IdleTime.Q THEN
				P4_SpodnyStoper.STAV.PoINIT:= TRUE;
				SC_P4_SpodnyStoper.ResetStep:= TRUE;
				SC_P4_SpodnyStoper.Step:= 100;
			END_IF

			//********************************************************Automatický režim****************************************************************************//
		100:
			SC_P4_SpodnyStoper.StepName:='100 - Automaticky Rezim - cakam na príchod paletky na stoper';
			SC_P4_SpodnyStoper.IdleTime.PT:= T#200ms;
			SC_P4_SpodnyStoper.AlarmTime.PT:= T#5s;

			SC_P4_SpodnyStoper.IdleTime.IN:= P4_SpodnyStoper.IN.PritomnostPaletky;

			IF P4_SpodnyStoper.KoniecCyklu THEN
				SC_P4_SpodnyStoper.ResetStep:= TRUE;
				SC_P4_SpodnyStoper.Step:= 0;
			ELSIF SC_P4_SpodnyStoper.IdleTime.Q THEN
				SC_P4_SpodnyStoper.ResetStep:= TRUE;
				SC_P4_SpodnyStoper.Step:= 101;
			END_IF

		101:
			SC_P4_SpodnyStoper.StepName:='101 - Automaticky Rezim - cakam na vyvezenie paletky na spodny stoper bunky 3';
			SC_P4_SpodnyStoper.IdleTime.PT:= T#2s;
			SC_P4_SpodnyStoper.AlarmTime.PT:= T#5s;

			SC_P4_SpodnyStoper.IdleTime.IN:= NOT P3_SpodnyStoper.IN.ZaplnenieDopravnika;

			IF P4_SpodnyStoper.KoniecCyklu THEN
				SC_P4_SpodnyStoper.ResetStep:= TRUE;
				SC_P4_SpodnyStoper.Step:= 0;
			ELSIF SC_P4_SpodnyStoper.IdleTime.Q AND P3_Dopravniky.STAV.PoINIT THEN
				SC_P4_SpodnyStoper.ResetStep:= TRUE;
				SC_P4_SpodnyStoper.Step:= 105;
			ELSIF NOT P4_SpodnyStoper.IN.PritomnostPaletky THEN
				SC_P4_SpodnyStoper.ResetStep:= TRUE;
				SC_P4_SpodnyStoper.Step:= 100;
			END_IF

		105:
			SC_P4_SpodnyStoper.StepName:='105 - Automaticky Rezim - vyvazam paletku na spodny stoper bunky 3';
			SC_P4_SpodnyStoper.IdleTime.PT:= T#200ms;
			SC_P4_SpodnyStoper.AlarmTime.PT:= T#10s;

			IF NOT SC_P4_SpodnyStoper.Switch1 THEN
				P4_SpodnyStoper.OUT.ZasunStoper:= TRUE;
				P4_SpodnyStoper.STAV.PrebiehaVyvezeniePaletky:= TRUE;
				SC_P4_SpodnyStoper.Switch1:= TRUE;
			END_IF

			IF NOT P4_SpodnyStoper.IN.PritomnostPaletky THEN
				P4_SpodnyStoper.OUT.ZasunStoper:= FALSE;
				P4_SpodnyStoper.STAV.PrebiehaVyvezeniePaletky:= FALSE;
				SC_P4_SpodnyStoper.ResetStep:= TRUE;
				SC_P4_SpodnyStoper.Step:= 100;
			END_IF

			//*******************************************************Manuálny režim*******************************************************************************//
		700:
			SC_P4_SpodnyStoper.StepName:='700 - Manualny Rezim';
			SC_P4_SpodnyStoper.IdleTime.PT:= T#8s;
			SC_P4_SpodnyStoper.AlarmTime.PT:= T#5s;

	END_CASE

END_PROGRAM

PROGRAM _EXIT
	(* Insert code here *)

END_PROGRAM
```

### Program Logical/Program/Pracovisko_4/P4_FunkcnyTestA (IEC)

#### Main.st - Init, cyclic, exit code
```iecst
PROGRAM _INIT

	P4_FunkcnyTestA.PAR.CisloPortuKlienta:= 1040;

END_PROGRAM

PROGRAM _CYCLIC

	//Volanie funkcie SequenceControl//
	SequenceControl(SC:= SC_P4_FunkcnyTestA);

	//Volanie podprogramov//
	OvlCentrovacky;
	OvlHornychKontaktov;
	OvlSpodnychKontaktov;
	IOLinkKomunikacia;
	COM_Tester;

	//Reset sekcie //
	IF P4_FunkcnyTestA.Reset THEN
		SC_P4_FunkcnyTestA.Step:= 0;
		P4_FunkcnyTestA.Reset:= FALSE;
	ELSIF NOT Safety.STAV.Linka_ZonaCS_AKTIVNA THEN
		SC_P4_FunkcnyTestA.Step:= 0;
	END_IF

	CASE SC_P4_FunkcnyTestA.Step OF

		0:
			SC_P4_FunkcnyTestA.StepName:='0 - Nulovanie';
			SC_OvlCentrovacky.Step:= 0;
			SC_OvlHornychKontaktov.Step:= 0;
			SC_OvlSpodnychKontaktov.Step:= 0;
			SC_OvlTesteraFT.Step:= 0;
			P4_FunkcnyTestA.Automat:= FALSE;
			P4_FunkcnyTestA.KoniecCyklu:= FALSE;
			P4_FunkcnyTestA.Manual:= FALSE;
			P4_FunkcnyTestA.STAV.PoINIT:= FALSE;
			P4_FunkcnyTestA.OUT.ZasunStoper:= FALSE;
			P4_FunkcnyTestA.OUT.KontaktyTestera_VYSUN:= FALSE;
			P4_FunkcnyTestA.OUT.OdpruzHornychKontaktov_VYSUN:= FALSE;
			P4_FunkcnyTestA.OUT.OdpruzHornychKontaktov_ZASUN:= TRUE;
			P4_FunkcnyTestA.OUT.PritlakPowerCP_VYSUN:= FALSE;
			P4_FunkcnyTestA.OUT.SpodneKontakty_VYSUN:= FALSE;
			P4_FunkcnyTestA.OUT.SpodneKontakty_ZASUN:= TRUE;
			P4_FunkcnyTestA.OUT.HorneKontakty_VYSUN:= FALSE;
			P4_FunkcnyTestA.OUT.HorneKontakty_ZASUN:= TRUE;
			P4_FunkcnyTestA.RFID_hlava.PrecitajChipRFID:= FALSE;
			P4_FunkcnyTestA.CMD.RR_ZatvorTester:= FALSE;
			P4_FunkcnyTestA.CMD.StartTestovania:= FALSE;
			P4_FunkcnyTestA.CMD.RR_VysunPruzenieKontaktov:= FALSE;
			P4_FunkcnyTestA.CMD.OpatovnyTest:= FALSE;
			P4_FunkcnyTestA.STAV.RR_SekvenciaTestera_BUSY:= FALSE;
			P4_FunkcnyTestA.STAV.PaletkaOznacena_NG:= FALSE;
			P34_Vizu.ZobrazHL1_FinalTestA:= FALSE;
			P3_ZdvizkaZaLeakTestA.STAV.PrebiehaVyvezeniePaletkyNaTratA:= FALSE;
			P4_FunkcnyTestA.STAV.PrebiehaVyvezeniePaletky:= FALSE;
			TestovaciKus:= FALSE;
			P4_FinalTestA_Taktime.IN.START_MeraniaCasu:= FALSE;
			P4_FinalTestA_Taktime.IN.START_MeraniaStratovehoCasu:= FALSE;

			PocetDopytovNaTester:= 0;

			IF Safety.STAV.Linka_ZonaCS_AKTIVNA AND
				Safety.STAV.P4_ZonaBunky_AKTIVNA AND
				P4_Pracovisko.STAV.HardwareBunky_OK AND
				NOT P4_Pracovisko.STAV.Porucha_ST1 AND
				NOT P4_Pracovisko.STAV.Porucha_ST2 AND
				NOT P4_Pracovisko.STAV.Porucha_ST3 AND
				NOT P4_Pracovisko.STAV.Porucha_ST4 AND
				NOT P4_Pracovisko.STAV.Porucha_ST5 AND
				NOT P4_Pracovisko.STAV.Porucha_ST6 THEN
				SC_P4_FunkcnyTestA.ResetStep:= TRUE;
				SC_P4_FunkcnyTestA.Step:= 1;
			END_IF

		1:
			SC_P4_FunkcnyTestA.StepName:='1 - Cakam na spustenie vyroby';
			P4_FunkcnyTestA.KoniecCyklu:= FALSE;
			IF P4_FunkcnyTestA.Automat THEN
				SC_P4_FunkcnyTestA.Step:= 2;
			ELSIF P4_FunkcnyTestA.Manual THEN
				SC_P4_FunkcnyTestA.Step:= 700;
			END_IF

			//********************************************************Inicializácia****************************************************************************//

		2:
			SC_P4_FunkcnyTestA.StepName:='2 - Inicializacia - cakam na spustenie inicializacie';
			SC_P4_FunkcnyTestA.IdleTime.PT:= T#500ms;
			SC_P4_FunkcnyTestA.AlarmTime.PT:= T#5s;

			SC_P4_FunkcnyTestA.IdleTime.IN:= TRUE;

			IF SC_P4_FunkcnyTestA.IdleTime.Q THEN
				SC_P4_FunkcnyTestA.ResetStep:= TRUE;
				SC_P4_FunkcnyTestA.Step:= 5;
			END_IF

		5:
			SC_P4_FunkcnyTestA.StepName:='5 - Inicializacia - zasunutie spodnych kontaktov';
			SC_P4_FunkcnyTestA.IdleTime.PT:= T#4s;
			SC_P4_FunkcnyTestA.AlarmTime.PT:= T#5s;

			IF NOT SC_P4_FunkcnyTestA.Switch1 THEN
				SpodneKontakty_ZASUN:= TRUE;
				SC_P4_FunkcnyTestA.Switch1:= TRUE;
			END_IF

			IF P4_FunkcnyTestA.IN.SpodneKontakty_ZASUNUTE THEN
				SC_P4_FunkcnyTestA.ResetStep:= TRUE;
				SC_P4_FunkcnyTestA.Step:= 8;
			END_IF

		8:
			SC_P4_FunkcnyTestA.StepName:='8 - Inicializacia - zasunutie hornych kontaktov';
			SC_P4_FunkcnyTestA.IdleTime.PT:= T#4s;
			SC_P4_FunkcnyTestA.AlarmTime.PT:= T#5s;

			IF NOT SC_P4_FunkcnyTestA.Switch1 THEN
				HorneKontakty_ZASUN:= TRUE;
				SC_P4_FunkcnyTestA.Switch1:= TRUE;
			END_IF

			IF P4_FunkcnyTestA.IN.HorneKontakty_ZASUNUTE THEN
				SC_P4_FunkcnyTestA.ResetStep:= TRUE;
				SC_P4_FunkcnyTestA.Step:= 10;
			END_IF

		10:
			SC_P4_FunkcnyTestA.StepName:='10 - Inicializacia - zasunutie cenrovacky';
			SC_P4_FunkcnyTestA.IdleTime.PT:= T#4s;
			SC_P4_FunkcnyTestA.AlarmTime.PT:= T#5s;

			IF NOT SC_P4_FunkcnyTestA.Switch1 THEN
				Centrovacku_ZASUN:= TRUE;
				SC_P4_FunkcnyTestA.Switch1:= TRUE;
			END_IF

			IF P4_FunkcnyTestA.IN.Centrovanie_ZASUNUTE THEN
				SC_P4_FunkcnyTestA.ResetStep:= TRUE;
				SC_P4_FunkcnyTestA.Step:= 13;
			END_IF

		13:
			SC_P4_FunkcnyTestA.StepName:='13 - Inicializacia - kontrola kontaktov Funkcneho testu';
			SC_P4_FunkcnyTestA.IdleTime.PT:= T#4s;
			SC_P4_FunkcnyTestA.AlarmTime.PT:= T#5s;

			IF Linka.PAR.ZvolenyModel = '4F' AND P4_FunkcnyTestA.IN.TypSpodnychKontaktov_4F THEN
				SC_P4_FunkcnyTestA.ResetStep:= TRUE;
				SC_P4_FunkcnyTestA.Step:= 15;
			ELSIF Linka.PAR.ZvolenyModel = '5F' AND P4_FunkcnyTestA.IN.TypSpodnychKontaktov_5F_5H THEN
				SC_P4_FunkcnyTestA.ResetStep:= TRUE;
				SC_P4_FunkcnyTestA.Step:= 15;
			ELSIF Linka.PAR.ZvolenyModel = '5H' AND P4_FunkcnyTestA.IN.TypSpodnychKontaktov_5F_5H THEN
				SC_P4_FunkcnyTestA.ResetStep:= TRUE;
				SC_P4_FunkcnyTestA.Step:= 15;
			ELSE
				P34_Alarmy[437]:= TRUE;
				P4_Pracovisko.STAV.Porucha_ST1:= TRUE;
			END_IF

		15:
			SC_P4_FunkcnyTestA.StepName:='15 - Inicializacia - hladanie paletky';
			SC_P4_FunkcnyTestA.IdleTime.PT:= T#5s;
			SC_P4_FunkcnyTestA.AlarmTime.PT:= T#5s;

			SC_P4_FunkcnyTestA.IdleTime.IN:= P4_Dopravniky.STAV.PoINIT;

			IF P4_FunkcnyTestA.RFID_hlava.PritomnostPaletky THEN
				SC_P4_FunkcnyTestA.ResetStep:= TRUE;
				SC_P4_FunkcnyTestA.Step:= 20;
			ELSIF SC_P4_FunkcnyTestA.IdleTime.Q THEN
				P4_FunkcnyTestA.STAV.PoINIT:= TRUE;
				SC_P4_FunkcnyTestA.ResetStep:= TRUE;
				SC_P4_FunkcnyTestA.Step:= 100;
			END_IF

		20:
			SC_P4_FunkcnyTestA.StepName:='20 - Inicializacia - precitanie cisla paletky';
			SC_P4_FunkcnyTestA.IdleTime.PT:= T#200ms;
			SC_P4_FunkcnyTestA.AlarmTime.PT:= T#5s;

			SC_P4_FunkcnyTestA.IdleTime.IN:= P4_FunkcnyTestA.RFID_hlava.PritomnostPaletky;

			IF SC_P4_FunkcnyTestA.IdleTime.Q AND NOT SC_P4_FunkcnyTestA.Switch1 THEN
				P4_FunkcnyTestA.RFID_hlava.PrecitajChipRFID:= TRUE;
				i:= 0;
				SC_P4_FunkcnyTestA.Switch1:= TRUE;
			END_IF

			IF P4_FunkcnyTestA.RFID_hlava.Stav_CitanieZapis_OK AND P4_FunkcnyTestA.RFID_hlava.PrecitaneCisloPaletky <> 0 THEN
				i:= P4_FunkcnyTestA.RFID_hlava.PrecitaneCisloPaletky;
				P4_FunkcnyTestA.RFID_hlava.PrecitajChipRFID:= FALSE;
				SC_P4_FunkcnyTestA.ResetStep:= TRUE;
				SC_P4_FunkcnyTestA.Step:= 23;
			END_IF

		23:
			SC_P4_FunkcnyTestA.StepName:='23 - Inicializacia - priradenie indexu paletky na zaklade precitanej hodnoty';
			SC_P4_FunkcnyTestA.IdleTime.PT:= T#200ms;
			SC_P4_FunkcnyTestA.AlarmTime.PT:= T#5s;

			IF i<> 0 THEN
				P4_FunkcnyTestA.PAR.CisloPaletky_STRING:= USINT_TO_STRING(i);
				Paletka[i].PAR.CisloPaletky:= USINT_TO_STRING(i);
				SC_P4_FunkcnyTestA.ResetStep:= TRUE;
				SC_P4_FunkcnyTestA.Step:= 30;
			ELSE
				P34_Alarmy[427]:= TRUE;
				P4_Pracovisko.STAV.Porucha_ST1:= TRUE;
			END_IF

		30:
			SC_P4_FunkcnyTestA.StepName:='30 - Inicializacia - kontrola stavu paletky';
			SC_P4_FunkcnyTestA.IdleTime.PT:= T#200ms;
			SC_P4_FunkcnyTestA.AlarmTime.PT:= T#5s;

			IF Paletka[i].STAV.StavPaletky = '' THEN
				Paletka[i].STAV.StavPaletky:= 'NG';
				SC_P4_FunkcnyTestA.ResetStep:= TRUE;
				SC_P4_FunkcnyTestA.Step:= 560;
			ELSIF Paletka[i].STAV.StavPaletky = 'PRECH' THEN
				P4_FunkcnyTestA.STAV.PoINIT:= TRUE;
				SC_P4_FunkcnyTestA.ResetStep:= TRUE;
				SC_P4_FunkcnyTestA.Step:= 560;
			ELSIF Paletka[i].STAV.StavPaletky = 'TEST' AND Paletka[i].STAV.CisloTestovacejStanice = 'ST_FT1,FT2' THEN
				TestovaciKus:= TRUE;
				P4_FunkcnyTestA.STAV.PoINIT:= TRUE;
				SC_P4_FunkcnyTestA.ResetStep:= TRUE;
				SC_P4_FunkcnyTestA.Step:= 110;
			ELSIF Paletka[i].STAV.StavPaletky = 'TEST' AND Paletka[i].STAV.CisloTestovacejStanice <> 'ST_FT1,FT2' THEN
				P4_FunkcnyTestA.STAV.PoINIT:= TRUE;
				SC_P4_FunkcnyTestA.ResetStep:= TRUE;
				SC_P4_FunkcnyTestA.Step:= 560;
			ELSIF Paletka[i].STAV.StavPaletky = 'REV' AND Paletka[i].STAV.CisloRevorkovejStanice = 'ST_FT1,FT2' THEN
				IF P4_FunkcnyTestA.STAV.Tester_ON THEN
					Paletka[i].STAV.StavPaletky:= 'OK';
					P4_FunkcnyTestA.STAV.PoINIT:= TRUE;
					SC_P4_FunkcnyTestA.ResetStep:= TRUE;
					SC_P4_FunkcnyTestA.Step:= 110;
				ELSE
					P4_FunkcnyTestA.STAV.PoINIT:= TRUE;
					SC_P4_FunkcnyTestA.ResetStep:= TRUE;
					SC_P4_FunkcnyTestA.Step:= 560;
				END_IF
			ELSIF Paletka[i].STAV.StavPaletky = 'REV' AND Paletka[i].STAV.CisloRevorkovejStanice <> 'ST_FT1,FT2' THEN
				P4_FunkcnyTestA.STAV.PoINIT:= TRUE;
				SC_P4_FunkcnyTestA.ResetStep:= TRUE;
				SC_P4_FunkcnyTestA.Step:= 560;
			ELSIF Paletka[i].STAV.StavPaletky = 'OK' THEN
				SC_P4_FunkcnyTestA.ResetStep:= TRUE;
				SC_P4_FunkcnyTestA.Step:= 33;
			ELSIF Paletka[i].STAV.StavPaletky = 'NG' THEN
				P4_FunkcnyTestA.STAV.PoINIT:= TRUE;
				SC_P4_FunkcnyTestA.ResetStep:= TRUE;
				SC_P4_FunkcnyTestA.Step:= 560;
			END_IF

		33:
			SC_P4_FunkcnyTestA.StepName:='33 - Inicializacia - kontrola ukonceneho HV testu';
			SC_P4_FunkcnyTestA.IdleTime.PT:= T#200ms;
			SC_P4_FunkcnyTestA.AlarmTime.PT:= T#5s;

			IF Paletka[i].STAV.FunkcnyTest_Ukonceny THEN
				P4_FunkcnyTestA.STAV.PoINIT:= TRUE;
				SC_P4_FunkcnyTestA.ResetStep:= TRUE;
				SC_P4_FunkcnyTestA.Step:= 560;
			ELSE
				P4_FunkcnyTestA.STAV.PoINIT:= TRUE;
				SC_P4_FunkcnyTestA.ResetStep:= TRUE;
				SC_P4_FunkcnyTestA.Step:= 110;
			END_IF

		//********************************************************Automatický režim****************************************************************************//

		100:
			SC_P4_FunkcnyTestA.StepName:='100 - Automaticky Rezim - cakam na príchod paletky na stoper';
			SC_P4_FunkcnyTestA.IdleTime.PT:= T#200ms;
			SC_P4_FunkcnyTestA.AlarmTime.PT:= T#5s;

			SC_P4_FunkcnyTestA.IdleTime.IN:= P4_FunkcnyTestA.RFID_hlava.PritomnostPaletky;

			IF P4_FunkcnyTestA.RFID_hlava.PritomnostPaletky THEN
				P3_ZdvizkaZaLeakTestA.STAV.PrebiehaVyvezeniePaletkyNaTratA:= FALSE;
			END_IF

			IF NOT SC_P4_FunkcnyTestA.Switch1 AND P4_FunkcnyTestA.RFID_hlava.PritomnostPaletky THEN
				P4_FinalTestA_Taktime.IN.START_MeraniaCasu:= TRUE;
				P4_FinalTestA_Taktime.IN.ZAPIS_MeraniaCasu:= TRUE;
				P4_FinalTestA_Taktime.IN.ZAPIS_StratovyCas:= TRUE;
				Buffer_11.Hodnota:= P4_FinalTestA_Taktime.OUT.StratoveSekundy;
				Buffer_11.ZapisHodnotu:= TRUE;
				SC_P4_FunkcnyTestA.Switch1:= TRUE;
			END_IF

			IF P4_FunkcnyTestA.KoniecCyklu THEN
				SC_P4_FunkcnyTestA.ResetStep:= TRUE;
				SC_P4_FunkcnyTestA.Step:= 0;
			ELSIF SC_P4_FunkcnyTestA.IdleTime.Q THEN
				SC_P4_FunkcnyTestA.ResetStep:= TRUE;
				SC_P4_FunkcnyTestA.Step:= 101;
			END_IF

		101:
			SC_P4_FunkcnyTestA.StepName:='101 - Automaticky Rezim - precitanie cisla paletky';
			SC_P4_FunkcnyTestA.IdleTime.PT:= T#200ms;
			SC_P4_FunkcnyTestA.AlarmTime.PT:= T#5s;
			SC_P4_FunkcnyTestA.IdleTime.IN:= TRUE;

			IF NOT SC_P4_FunkcnyTestA.Switch1 THEN
				P4_FunkcnyTestA.RFID_hlava.PrecitajChipRFID:= TRUE;
				i:= 0;
				SC_P4_FunkcnyTestA.Switch1:= TRUE;
			END_IF

			IF P4_FunkcnyTestA.RFID_hlava.Stav_CitanieZapis_OK AND P4_FunkcnyTestA.RFID_hlava.PrecitaneCisloPaletky <> 0 THEN
				i:= P4_FunkcnyTestA.RFID_hlava.PrecitaneCisloPaletky;
				P4_FunkcnyTestA.RFID_hlava.PrecitajChipRFID:= FALSE;
				SC_P4_FunkcnyTestA.ResetStep:= TRUE;
				SC_P4_FunkcnyTestA.Step:= 102;
			END_IF

		102:
			SC_P4_FunkcnyTestA.StepName:='102 - Automaticky Rezim - priradenie indexu paletky na zaklade precitanej hodnoty';
			SC_P4_FunkcnyTestA.IdleTime.PT:= T#200ms;
			SC_P4_FunkcnyTestA.AlarmTime.PT:= T#5s;

			IF i<> 0 THEN
				P4_FunkcnyTestA.PAR.CisloPaletky_STRING:= USINT_TO_STRING(i);
				Paletka[i].PAR.CisloPaletky:= USINT_TO_STRING(i);
				SC_P4_FunkcnyTestA.ResetStep:= TRUE;
				SC_P4_FunkcnyTestA.Step:= 103;
			ELSE
				P34_Alarmy[427]:= TRUE;
				P4_Pracovisko.STAV.Porucha_ST1:= TRUE;
			END_IF

		103:
			SC_P4_FunkcnyTestA.StepName:='103 - Automaticky Rezim - kontrola stavu paletky';
			SC_P4_FunkcnyTestA.IdleTime.PT:= T#200ms;
			SC_P4_FunkcnyTestA.AlarmTime.PT:= T#5s;

			IF Paletka[i].STAV.StavPaletky = '' THEN
				Paletka[i].STAV.StavPaletky:= 'NG';
				SC_P4_FunkcnyTestA.ResetStep:= TRUE;
				SC_P4_FunkcnyTestA.Step:= 560;
			ELSIF Paletka[i].STAV.StavPaletky = 'PRECH' THEN
				SC_P4_FunkcnyTestA.ResetStep:= TRUE;
				SC_P4_FunkcnyTestA.Step:= 560;
			ELSIF Paletka[i].STAV.StavPaletky = 'TEST' AND Paletka[i].STAV.CisloTestovacejStanice = 'ST_FT1,FT2' THEN
				TestovaciKus:= TRUE;
				SC_P4_FunkcnyTestA.ResetStep:= TRUE;
				SC_P4_FunkcnyTestA.Step:= 110;
			ELSIF Paletka[i].STAV.StavPaletky = 'TEST' AND Paletka[i].STAV.CisloTestovacejStanice <> 'ST_FT1,FT2' THEN
				SC_P4_FunkcnyTestA.ResetStep:= TRUE;
				SC_P4_FunkcnyTestA.Step:= 560;
			ELSIF Paletka[i].STAV.StavPaletky = 'REV' AND Paletka[i].STAV.CisloRevorkovejStanice = 'ST_FT1,FT2' THEN
				IF P4_FunkcnyTestA.STAV.Tester_ON THEN
					Paletka[i].STAV.StavPaletky:= 'OK';
					SC_P4_FunkcnyTestA.ResetStep:= TRUE;
					SC_P4_FunkcnyTestA.Step:= 110;
				ELSE
					SC_P4_FunkcnyTestA.ResetStep:= TRUE;
					SC_P4_FunkcnyTestA.Step:= 560;
				END_IF
			ELSIF Paletka[i].STAV.StavPaletky = 'REV' AND Paletka[i].STAV.CisloRevorkovejStanice <> 'ST_FT1,FT2' THEN
				SC_P4_FunkcnyTestA.ResetStep:= TRUE;
				SC_P4_FunkcnyTestA.Step:= 560;
			ELSIF Paletka[i].STAV.StavPaletky = 'OK' THEN
				SC_P4_FunkcnyTestA.ResetStep:= TRUE;
				SC_P4_FunkcnyTestA.Step:= 110;
			ELSIF Paletka[i].STAV.StavPaletky = 'NG' THEN
				SC_P4_FunkcnyTestA.ResetStep:= TRUE;
				SC_P4_FunkcnyTestA.Step:= 560;
			END_IF

		//Zatvorenie Funkčného testera//

		110:
			SC_P4_FunkcnyTestA.StepName:='110 - Automaticky Rezim - zacentrovanie paletky';
			SC_P4_FunkcnyTestA.IdleTime.PT:= T#200ms;
			SC_P4_FunkcnyTestA.AlarmTime.PT:= T#5s;

			IF NOT SC_P4_FunkcnyTestA.Switch1 THEN
				Centrovacku_VYSUN:= TRUE;
				SC_P4_FunkcnyTestA.Switch1:= TRUE;
			END_IF

			IF P4_FunkcnyTestA.IN.Centrovanie_VYSUNUTE THEN
				SC_P4_FunkcnyTestA.ResetStep:= TRUE;
				SC_P4_FunkcnyTestA.Step:= 113;
			END_IF

		113:
			SC_P4_FunkcnyTestA.StepName:='113 - Automaticky Rezim - vysunutie pruzenia hornych kontaktov';
			SC_P4_FunkcnyTestA.IdleTime.PT:= T#500ms;
			SC_P4_FunkcnyTestA.AlarmTime.PT:= T#5s;

			IF NOT SC_P4_FunkcnyTestA.Switch1 THEN
				P4_FunkcnyTestA.OUT.OdpruzHornychKontaktov_ZASUN:= FALSE;
				P4_FunkcnyTestA.OUT.OdpruzHornychKontaktov_VYSUN:= TRUE;
				SC_P4_FunkcnyTestA.IdleTime.IN:= TRUE;
				SC_P4_FunkcnyTestA.Switch1:= TRUE;
			END_IF

			IF SC_P4_FunkcnyTestA.IdleTime.Q THEN
				SC_P4_FunkcnyTestA.ResetStep:= TRUE;
				SC_P4_FunkcnyTestA.Step:= 115;
			END_IF

		115:
			SC_P4_FunkcnyTestA.StepName:='115 - Automaticky Rezim - vysunutie hornych kontaktov';
			SC_P4_FunkcnyTestA.IdleTime.PT:= T#200ms;
			SC_P4_FunkcnyTestA.AlarmTime.PT:= T#5s;

			IF NOT SC_P4_FunkcnyTestA.Switch1 THEN
				HorneKontakty_VYSUN:= TRUE;
				SC_P4_FunkcnyTestA.Switch1:= TRUE;
			END_IF

			IF P4_FunkcnyTestA.IN.HorneKontakty_VYSUNUTE THEN
				SC_P4_FunkcnyTestA.ResetStep:= TRUE;
				SC_P4_FunkcnyTestA.Step:= 118;
			END_IF

		118:
			SC_P4_FunkcnyTestA.StepName:='118 - Automaticky Rezim - vysunutie spodnych kontaktov';
			SC_P4_FunkcnyTestA.IdleTime.PT:= T#200ms;
			SC_P4_FunkcnyTestA.AlarmTime.PT:= T#5s;

			IF NOT SC_P4_FunkcnyTestA.Switch1 THEN
				SpodneKontakty_VYSUN:= TRUE;
				SC_P4_FunkcnyTestA.Switch1:= TRUE;
			END_IF

			IF P4_FunkcnyTestA.IN.SpodneKontakty_VYSUNUTE THEN
				SC_P4_FunkcnyTestA.ResetStep:= TRUE;
				SC_P4_FunkcnyTestA.Step:= 120;
			END_IF

		120:
			SC_P4_FunkcnyTestA.StepName:='120 - Automaticky Rezim - pritlacenie kontaktov testera';
			SC_P4_FunkcnyTestA.IdleTime.PT:= T#1s;
			SC_P4_FunkcnyTestA.AlarmTime.PT:= T#5s;

			P4_FunkcnyTestA.OUT.KontaktyTestera_VYSUN:= TRUE;
			SC_P4_FunkcnyTestA.IdleTime.IN:= TRUE;

			IF SC_P4_FunkcnyTestA.IdleTime.Q THEN
				IF P4_FunkcnyTestA.Manual THEN
					IF NOT P4_FunkcnyTestA.CMD.RR_ZatvorTester THEN
						SC_P4_FunkcnyTestA.ResetStep:= TRUE;
						SC_P4_FunkcnyTestA.Step:= 140;
					END_IF
				ELSE
					SC_P4_FunkcnyTestA.ResetStep:= TRUE;
					SC_P4_FunkcnyTestA.Step:= 130;
				END_IF
			END_IF

		130:
			SC_P4_FunkcnyTestA.StepName:='130 - Automaticky Rezim - spustenie testera';
			SC_P4_FunkcnyTestA.IdleTime.PT:= T#2s;
			SC_P4_FunkcnyTestA.AlarmTime.PT:= T#5s;

			SC_P4_FunkcnyTestA.IdleTime.IN:= TRUE;

			IF Linka.KOM_Panatrace_OFF THEN
				IF SC_P4_FunkcnyTestA.IdleTime.Q THEN
					SC_P4_FunkcnyTestA.ResetStep:= TRUE;
					SC_P4_FunkcnyTestA.Step:= 140;
				END_IF
			ELSE
				P4_FunkcnyTestA.STAV.Vysledok_FV_Testu:= '';
				P4_FunkcnyTestA.CMD.StartTestovania:= TRUE;
				P4_FinalTestA_Taktime.IN.START_MeraniaStratovehoCasu:= TRUE;
				SC_P4_FunkcnyTestA.ResetStep:= TRUE;
				SC_P4_FunkcnyTestA.Step:= 133;
			END_IF

		133:
			SC_P4_FunkcnyTestA.StepName:='133 - Automaticky Rezim - cakam na ukoncenie HV testu';
			SC_P4_FunkcnyTestA.IdleTime.PT:= T#1s;
			SC_P4_FunkcnyTestA.AlarmTime.PT:= T#5s;

			IF P4_FunkcnyTestA.STAV.TestovanieUkoncene THEN
				P4_FinalTestA_Taktime.IN.START_MeraniaStratovehoCasu:= FALSE;
				Paletka[i].STAV.FunkcnyTest_Ukonceny:= TRUE;
				P4_FunkcnyTestA.CMD.StartTestovania:= FALSE;
				IF Paletka[i].STAV.StavPaletky = 'TEST' THEN
					SC_P4_FunkcnyTestA.ResetStep:= TRUE;
					SC_P4_FunkcnyTestA.Step:= 135;
				ELSE
					IF P4_FunkcnyTestA.STAV.Vysledok_FV_Testu = 'OK' THEN
						Paletka[i].STAV.StavPaletky:= 'OK';
					ELSIF P4_FunkcnyTestA.STAV.Vysledok_FV_Testu = 'NG' THEN
						Paletka[i].STAV.StavPaletky:= 'NG';
					END_IF
					SC_P4_FunkcnyTestA.ResetStep:= TRUE;
					SC_P4_FunkcnyTestA.Step:= 135;
				END_IF
			ELSIF P4_FunkcnyTestA.STAV.TesterNeodpoveda THEN
				P4_FunkcnyTestA.CMD.StartTestovania:= FALSE;
				SC_P4_FunkcnyTestA.ResetStep:= TRUE;
				SC_P4_FunkcnyTestA.Step:= 134;
			END_IF

		134:
			SC_P4_FunkcnyTestA.StepName:='134 - Automaticky Rezim - zobrazenie hlasenia tester neodpoveda';
			SC_P4_FunkcnyTestA.IdleTime.PT:= T#1s;
			SC_P4_FunkcnyTestA.AlarmTime.PT:= T#5s;

			P34_Vizu.ZobrazHL1_FinalTestA:= TRUE;

			IF P4_FunkcnyTestA.CMD.OpatovnyTest THEN
				P4_FunkcnyTestA.CMD.OpatovnyTest:= FALSE;
				P34_Vizu.ZobrazHL1_FinalTestA:= FALSE;
				IF P4_FunkcnyTestA.PAR.CisloPortuKlienta < 1049 THEN
					P4_FunkcnyTestA.PAR.CisloPortuKlienta:= P4_FunkcnyTestA.PAR.CisloPortuKlienta + 1;
				ELSE
					P4_FunkcnyTestA.PAR.CisloPortuKlienta:= 1040;
				END_IF
				SC_P4_FunkcnyTestA.ResetStep:= TRUE;
				SC_P4_FunkcnyTestA.Step:= 130;
			ELSIF P4_FunkcnyTestA.STAV.PaletkaOznacena_NG THEN
				P4_FunkcnyTestA.STAV.PaletkaOznacena_NG:= FALSE;
				P34_Vizu.ZobrazHL1_FinalTestA:= FALSE;
				Paletka[i].STAV.StavPaletky:= 'NG';
				SC_P4_FunkcnyTestA.ResetStep:= TRUE;
				SC_P4_FunkcnyTestA.Step:= 135;
			END_IF

		135:
			SC_P4_FunkcnyTestA.StepName:='135 - Automaticky Rezim - cakam na zrusenie signalu Funkcny test ukonceny';
			SC_P4_FunkcnyTestA.IdleTime.PT:= T#1s;
			SC_P4_FunkcnyTestA.AlarmTime.PT:= T#5s;

			IF NOT P4_FunkcnyTestA.STAV.TestovanieUkoncene THEN
				SC_P4_FunkcnyTestA.ResetStep:= TRUE;
				SC_P4_FunkcnyTestA.Step:= 140;
			END_IF

			//Otvorenie Funkcneho testera//

		140:
			SC_P4_FunkcnyTestA.StepName:='140 - Automaticky Rezim - zasunutie pritlacenia kontaktov testera';
			SC_P4_FunkcnyTestA.IdleTime.PT:= T#1s;
			SC_P4_FunkcnyTestA.AlarmTime.PT:= T#5s;

			P4_FunkcnyTestA.OUT.KontaktyTestera_VYSUN:= FALSE;
			SC_P4_FunkcnyTestA.IdleTime.IN:= TRUE;

			IF SC_P4_FunkcnyTestA.IdleTime.Q THEN
				SC_P4_FunkcnyTestA.ResetStep:= TRUE;
				SC_P4_FunkcnyTestA.Step:= 143;
			END_IF

		143:
			SC_P4_FunkcnyTestA.StepName:='143 - Automaticky Rezim - zasunutie spodnych kontaktov';
			SC_P4_FunkcnyTestA.IdleTime.PT:= T#200ms;
			SC_P4_FunkcnyTestA.AlarmTime.PT:= T#5s;

			IF NOT SC_P4_FunkcnyTestA.Switch1 THEN
				P4_FunkcnyTestA.OUT.PritlakPowerCP_VYSUN:= TRUE;
				SpodneKontakty_ZASUN:= TRUE;
				SC_P4_FunkcnyTestA.Switch1:= TRUE;
			END_IF

			IF P4_FunkcnyTestA.IN.SpodneKontakty_ZASUNUTE THEN
				SC_P4_FunkcnyTestA.ResetStep:= TRUE;
				SC_P4_FunkcnyTestA.Step:= 145;
			END_IF

		145:
			SC_P4_FunkcnyTestA.StepName:='145 - Automaticky Rezim - zasunutie hornych kontaktov';
			SC_P4_FunkcnyTestA.IdleTime.PT:= T#200ms;
			SC_P4_FunkcnyTestA.AlarmTime.PT:= T#5s;

			IF NOT SC_P4_FunkcnyTestA.Switch1 THEN
				HorneKontakty_ZASUN:= TRUE;
				SC_P4_FunkcnyTestA.Switch1:= TRUE;
			END_IF

			IF P4_FunkcnyTestA.IN.HorneKontakty_ZASUNUTE THEN
				P4_FunkcnyTestA.OUT.PritlakPowerCP_VYSUN:= FALSE;
				SC_P4_FunkcnyTestA.ResetStep:= TRUE;
				SC_P4_FunkcnyTestA.Step:= 148;
			END_IF

		148:
			SC_P4_FunkcnyTestA.StepName:='148 - Automaticky Rezim - zasunutie pruzenia hornych kontaktov';
			SC_P4_FunkcnyTestA.IdleTime.PT:= T#500ms;
			SC_P4_FunkcnyTestA.AlarmTime.PT:= T#5s;

			IF NOT SC_P4_FunkcnyTestA.Switch1 THEN
				P4_FunkcnyTestA.OUT.OdpruzHornychKontaktov_VYSUN:= FALSE;
				P4_FunkcnyTestA.OUT.OdpruzHornychKontaktov_ZASUN:= TRUE;
				SC_P4_FunkcnyTestA.IdleTime.IN:= TRUE;
			END_IF

			IF SC_P4_FunkcnyTestA.IdleTime.Q THEN
				SC_P4_FunkcnyTestA.ResetStep:= TRUE;
				SC_P4_FunkcnyTestA.Step:= 150;
			END_IF

		150:
			SC_P4_FunkcnyTestA.StepName:='150 - Automaticky Rezim - odcentrovanie paletky';
			SC_P4_FunkcnyTestA.IdleTime.PT:= T#200ms;
			SC_P4_FunkcnyTestA.AlarmTime.PT:= T#5s;

			IF NOT SC_P4_FunkcnyTestA.Switch1 THEN
				Centrovacku_ZASUN:= TRUE;
				SC_P4_FunkcnyTestA.Switch1:= TRUE;
			END_IF

			IF P4_FunkcnyTestA.IN.Centrovanie_ZASUNUTE THEN
				IF P4_FunkcnyTestA.Manual THEN
					P4_FunkcnyTestA.STAV.RR_SekvenciaTestera_BUSY:= FALSE;
					SC_P4_FunkcnyTestA.ResetStep:= TRUE;
					SC_P4_FunkcnyTestA.Step:= 700;
				ELSE
					SC_P4_FunkcnyTestA.ResetStep:= TRUE;
					SC_P4_FunkcnyTestA.Step:= 560;
				END_IF
			END_IF

		//***************************Vyvezenie paletky**********************************************//

		560:
			SC_P4_FunkcnyTestA.StepName:='560 - Automaticky Rezim - cakam na vyvezenie na zdvižku za Funkcnym Testom A';
			SC_P4_FunkcnyTestA.IdleTime.PT:= T#200ms;
			SC_P4_FunkcnyTestA.AlarmTime.PT:= T#5s;

			IF P4_FunkcnyTestA.KoniecCyklu THEN
				SC_P4_FunkcnyTestA.ResetStep:= TRUE;
				SC_P4_FunkcnyTestA.Step:= 0;
			ELSIF NOT P4_ZdvizkaZaFunkcTestA.IN.PritomnostPaletky AND
				SC_P4_ZdvizkaZaFunkcTestA.Step = 100 AND
				NOT P4_FunkcnyTestA.STAV.PrebiehaVyvezeniePaletky AND
				NOT P4_ZdvizkaZaFunkcTestB.STAV.PrebiehaVyvezeniePaletky AND
				P4_ZdvizkaZaFunkcTestA.STAV.PoINIT AND
				P4_ZdvizkaZaFunkcTestA.IN.Zdvizka_StrednaPoloha AND
				P4_ZdvizkaZaFunkcTestB.STAV.PoINIT THEN
				P4_FunkcnyTestA.OUT.ZasunStoper:= TRUE;
				P4_FunkcnyTestA.STAV.PrebiehaVyvezeniePaletky:= TRUE;
				SC_P4_FunkcnyTestA.ResetStep:= TRUE;
				SC_P4_FunkcnyTestA.Step:= 561;
			END_IF

		561:
			SC_P4_FunkcnyTestA.StepName:='561 - Automaticky Rezim - ukoncenie vyvazania na zdvižku za Funkcnym Testom A';
			SC_P4_FunkcnyTestA.IdleTime.PT:= T#200ms;
			SC_P4_FunkcnyTestA.AlarmTime.PT:= T#10s;

			SC_P4_FunkcnyTestA.AlarmTime.IN:= P4_FunkcnyTestA.RFID_hlava.PritomnostPaletky;
			SC_P4_FunkcnyTestA.IdleTime.IN:= NOT P4_FunkcnyTestA.RFID_hlava.PritomnostPaletky;

			IF NOT P4_FunkcnyTestA.RFID_hlava.PritomnostPaletky THEN
				TestovaciKus:= FALSE;
				Paletka[i].PAR.StavPowerCP:= '';
				Paletka[i].STAV.Komunikacia_DONE:= FALSE;
				Paletka[i].STAV.OdoslanieFotiek_DONE:= FALSE;
				P4_FunkcnyTestA.OUT.ZasunStoper:= FALSE;
				SC_P4_FunkcnyTestA.ResetStep:= TRUE;
				SC_P4_FunkcnyTestA.Step:= 100;
			ELSIF SC_P4_FunkcnyTestA.AlarmTime.Q THEN
				P34_Alarmy[450]:= TRUE;
				P4_Pracovisko.STAV.Porucha_ST1:= TRUE;
			END_IF

		//*******************************************************Manuálny režim*******************************************************************************//
		700:
			SC_P4_FunkcnyTestA.StepName:='700 - Manualny Rezim';
			SC_P4_FunkcnyTestA.IdleTime.PT:= T#8s;
			SC_P4_FunkcnyTestA.AlarmTime.PT:= T#5s;

			//Sekvencia zatvárania testera//
			IF P4_FunkcnyTestA.CMD.RR_ZatvorTester THEN
				P4_FunkcnyTestA.STAV.RR_SekvenciaTestera_BUSY:= TRUE;
				SC_P4_FunkcnyTestA.ResetStep:= TRUE;
				SC_P4_FunkcnyTestA.Step:= 110;
			END_IF

			//Ovládanie zdvižky//
			IF P4_FunkcnyTestA.CMD.RR_VysunCentrovanie THEN
				P4_FunkcnyTestA.OUT.Centrovanie_VYSUN:= TRUE;
				P4_FunkcnyTestA.OUT.Centrovanie_ZASUN:= FALSE;
			ELSE
				P4_FunkcnyTestA.OUT.Centrovanie_VYSUN:= FALSE;
				P4_FunkcnyTestA.OUT.Centrovanie_ZASUN:= TRUE;
			END_IF

			//Ovládanie pruženia horných kontaktov//
			IF P4_FunkcnyTestA.CMD.RR_VysunPruzenieKontaktov THEN
				P4_FunkcnyTestA.OUT.OdpruzHornychKontaktov_ZASUN:= FALSE;
				P4_FunkcnyTestA.OUT.OdpruzHornychKontaktov_VYSUN:= TRUE;
			ELSE
				P4_FunkcnyTestA.OUT.OdpruzHornychKontaktov_ZASUN:= TRUE;
				P4_FunkcnyTestA.OUT.OdpruzHornychKontaktov_VYSUN:= FALSE;
			END_IF

	END_CASE

END_PROGRAM

PROGRAM _EXIT
	(* Insert code here *)

END_PROGRAM
```

#### Variables.var - Local variables
```iecst
VAR
	SC_OvlCentrovacky : SequenceControlTyp;
	Centrovacku_VYSUN : BOOL;
	Centrovacku_ZASUN : BOOL;
	SC_OvlSpodnychKontaktov : SequenceControlTyp;
	SpodneKontakty_VYSUN : BOOL;
	SpodneKontakty_ZASUN : BOOL;
	SC_OvlHornychKontaktov : SequenceControlTyp;
	HorneKontakty_VYSUN : BOOL;
	HorneKontakty_ZASUN : BOOL;
	i : USINT;
	TestovaciKus : BOOL := 0;
	SC_OvlTesteraFT : SequenceControlTyp;
	SKTcpClientTester_0 : SKTcpClientTester;
	dataStr : STRING[32];
	PocetDopytovNaTester : USINT := 0;
	Cas_FunkcnyTestA : TON;
	NameranyCasFunkcnehoTestuA : TIME := T#0S;
END_VAR
```

#### IOLinkKomunikacia.st
```iecst
ACTION IOLinkKomunikacia:

	//RFID snímač paletky//
	P4_FunkcnyTestA.RFID_hlava();

END_ACTION
```

#### OvlCentrovacky.st
```iecst
ACTION OvlCentrovacky:

	//Volanie funkcie SequenceControl//
	SequenceControl(SC:= SC_OvlCentrovacky);

	CASE SC_OvlCentrovacky.Step OF

		0:
			SC_OvlCentrovacky.StepName:= '0 - Nulovanie';
			Centrovacku_VYSUN:= FALSE;
			Centrovacku_ZASUN:= FALSE;

			IF SC_P4_FunkcnyTestA.Step <> 0 THEN
				SC_OvlCentrovacky.ResetStep:= TRUE;
				SC_OvlCentrovacky.Step:= 1;
			END_IF

		1:
			SC_OvlCentrovacky.StepName:= '1 - Rozhodnutie o cinnosti';
			IF Centrovacku_VYSUN THEN
				SC_OvlCentrovacky.Step:= 10;
			ELSIF Centrovacku_ZASUN THEN
				SC_OvlCentrovacky.Step:= 20;
			END_IF

		10:
			SC_OvlCentrovacky.StepName:= '10 - Vysunutie centrovacky';
			SC_OvlCentrovacky.IdleTime.PT:= T#3s;
			SC_OvlCentrovacky.AlarmTime.PT:= T#6s;

			IF P4_FunkcnyTestA.Automat THEN
				SC_OvlCentrovacky.AlarmTime.IN:= TRUE;
			ELSE
				SC_OvlCentrovacky.IdleTime.IN:= TRUE;
			END_IF

			IF NOT SC_OvlCentrovacky.Switch1 THEN
				P4_FunkcnyTestA.OUT.Centrovanie_ZASUN:= FALSE;
                P4_FunkcnyTestA.OUT.Centrovanie_VYSUN:= TRUE;
				SC_OvlCentrovacky.Switch1:= TRUE;
			END_IF

			IF P4_FunkcnyTestA.IN.Centrovanie_VYSUNUTE OR SC_OvlCentrovacky.IdleTime.Q THEN
				SC_OvlCentrovacky.ResetStep:= TRUE;
				SC_OvlCentrovacky.Step:= 0;
			ELSIF SC_OvlCentrovacky.AlarmTime.Q THEN
				P34_Alarmy[400]:= TRUE;
				P4_Pracovisko.STAV.Porucha_ST1:= TRUE;
			END_IF

		20:
			SC_OvlCentrovacky.StepName:= '20 - Zasunutie centrovacky';
			SC_OvlCentrovacky.IdleTime.PT:= T#3s;
			SC_OvlCentrovacky.AlarmTime.PT:= T#6s;

			IF P4_FunkcnyTestA.Automat THEN
				SC_OvlCentrovacky.AlarmTime.IN:= TRUE;
			ELSE
				SC_OvlCentrovacky.IdleTime.IN:= TRUE;
			END_IF

			IF NOT SC_OvlCentrovacky.Switch1 THEN
				P4_FunkcnyTestA.OUT.Centrovanie_VYSUN:= FALSE;
                P4_FunkcnyTestA.OUT.Centrovanie_ZASUN:= TRUE;
				SC_OvlCentrovacky.Switch1:= TRUE;
			END_IF

			IF P4_FunkcnyTestA.IN.Centrovanie_ZASUNUTE OR SC_OvlCentrovacky.IdleTime.Q THEN
				SC_OvlCentrovacky.ResetStep:= TRUE;
				SC_OvlCentrovacky.Step:= 0;
			ELSIF SC_OvlCentrovacky.AlarmTime.Q THEN
				P34_Alarmy[401]:= TRUE;
				P4_Pracovisko.STAV.Porucha_ST1:= TRUE;
			END_IF

	END_CASE

END_ACTION
```

#### OvlSpodnychKontaktov.st
```iecst
ACTION OvlSpodnychKontaktov:

	//Volanie funkcie SequenceControl//
	SequenceControl(SC:= SC_OvlSpodnychKontaktov);

	CASE SC_OvlSpodnychKontaktov.Step OF

		0:
			SC_OvlSpodnychKontaktov.StepName:= '0 - Nulovanie';
			SpodneKontakty_VYSUN:= FALSE;
			SpodneKontakty_ZASUN:= FALSE;

			IF SC_P4_FunkcnyTestA.Step <> 0 THEN
				SC_OvlSpodnychKontaktov.ResetStep:= TRUE;
				SC_OvlSpodnychKontaktov.Step:= 1;
			END_IF

		1:
			SC_OvlSpodnychKontaktov.StepName:= '1 - Rozhodnutie o cinnosti';
			IF SpodneKontakty_VYSUN THEN
				SC_OvlSpodnychKontaktov.Step:= 10;
			ELSIF SpodneKontakty_ZASUN THEN
				SC_OvlSpodnychKontaktov.Step:= 20;
			END_IF

		10:
			SC_OvlSpodnychKontaktov.StepName:= '10 - Vysunutie spodnych kontaktov';
			SC_OvlSpodnychKontaktov.IdleTime.PT:= T#3s;
			SC_OvlSpodnychKontaktov.AlarmTime.PT:= T#6s;

			IF P4_FunkcnyTestA.Automat THEN
				SC_OvlSpodnychKontaktov.AlarmTime.IN:= TRUE;
			ELSE
				SC_OvlSpodnychKontaktov.IdleTime.IN:= TRUE;
			END_IF

			IF NOT SC_OvlSpodnychKontaktov.Switch1 THEN
				P4_FunkcnyTestA.OUT.SpodneKontakty_ZASUN:= FALSE;
                P4_FunkcnyTestA.OUT.SpodneKontakty_VYSUN:= TRUE;
				SC_OvlSpodnychKontaktov.Switch1:= TRUE;
			END_IF

			IF P4_FunkcnyTestA.IN.SpodneKontakty_VYSUNUTE OR SC_OvlSpodnychKontaktov.IdleTime.Q THEN
				SC_OvlSpodnychKontaktov.ResetStep:= TRUE;
				SC_OvlSpodnychKontaktov.Step:= 0;
			ELSIF SC_OvlSpodnychKontaktov.AlarmTime.Q THEN
				P34_Alarmy[421]:= TRUE;
				P4_Pracovisko.STAV.Porucha_ST1:= TRUE;
			END_IF

		20:
			SC_OvlSpodnychKontaktov.StepName:= '20 - Zasunutie spodnych kontaktov';
			SC_OvlSpodnychKontaktov.IdleTime.PT:= T#3s;
			SC_OvlSpodnychKontaktov.AlarmTime.PT:= T#6s;

			IF P4_FunkcnyTestA.Automat THEN
				SC_OvlSpodnychKontaktov.AlarmTime.IN:= TRUE;
			ELSE
				SC_OvlSpodnychKontaktov.IdleTime.IN:= TRUE;
			END_IF

			IF NOT SC_OvlSpodnychKontaktov.Switch1 THEN
				P4_FunkcnyTestA.OUT.SpodneKontakty_VYSUN:= FALSE;
                P4_FunkcnyTestA.OUT.SpodneKontakty_ZASUN:= TRUE;
				SC_OvlSpodnychKontaktov.Switch1:= TRUE;
			END_IF

			IF P4_FunkcnyTestA.IN.SpodneKontakty_ZASUNUTE OR SC_OvlSpodnychKontaktov.IdleTime.Q THEN
				SC_OvlSpodnychKontaktov.ResetStep:= TRUE;
				SC_OvlSpodnychKontaktov.Step:= 0;
			ELSIF SC_OvlSpodnychKontaktov.AlarmTime.Q THEN
				P34_Alarmy[422]:= TRUE;
				P4_Pracovisko.STAV.Porucha_ST1:= TRUE;
			END_IF

	END_CASE

END_ACTION
```

#### OvlHornychKontaktov.st
```iecst
ACTION OvlHornychKontaktov:

	//Volanie funkcie SequenceControl//
	SequenceControl(SC:= SC_OvlHornychKontaktov);

	CASE SC_OvlHornychKontaktov.Step OF

		0:
			SC_OvlHornychKontaktov.StepName:= '0 - Nulovanie';
			HorneKontakty_VYSUN:= FALSE;
			HorneKontakty_ZASUN:= FALSE;

			IF SC_P4_FunkcnyTestA.Step <> 0 THEN
				SC_OvlHornychKontaktov.ResetStep:= TRUE;
				SC_OvlHornychKontaktov.Step:= 1;
			END_IF

		1:
			SC_OvlHornychKontaktov.StepName:= '1 - Rozhodnutie o cinnosti';
			IF HorneKontakty_VYSUN THEN
				SC_OvlHornychKontaktov.Step:= 10;
			ELSIF HorneKontakty_ZASUN THEN
				SC_OvlHornychKontaktov.Step:= 20;
			END_IF

		10:
			SC_OvlHornychKontaktov.StepName:= '10 - Vysunutie hornych kontaktov';
			SC_OvlHornychKontaktov.IdleTime.PT:= T#3s;
			SC_OvlHornychKontaktov.AlarmTime.PT:= T#6s;

			IF P4_FunkcnyTestA.Automat THEN
				SC_OvlHornychKontaktov.AlarmTime.IN:= TRUE;
			ELSE
				SC_OvlHornychKontaktov.IdleTime.IN:= TRUE;
			END_IF

			IF NOT SC_OvlHornychKontaktov.Switch1 THEN
				P4_FunkcnyTestA.OUT.HorneKontakty_ZASUN:= FALSE;
				P4_FunkcnyTestA.OUT.HorneKontakty_VYSUN:= TRUE;
				SC_OvlHornychKontaktov.Switch1:= TRUE;
			END_IF

			IF P4_FunkcnyTestA.IN.HorneKontakty_VYSUNUTE OR SC_OvlHornychKontaktov.IdleTime.Q THEN
				SC_OvlHornychKontaktov.ResetStep:= TRUE;
				SC_OvlHornychKontaktov.Step:= 0;
			ELSIF SC_OvlHornychKontaktov.AlarmTime.Q THEN
				P34_Alarmy[419]:= TRUE;
				P4_Pracovisko.STAV.Porucha_ST1:= TRUE;
			END_IF

		20:
			SC_OvlHornychKontaktov.StepName:= '20 - Zasunutie hornych kontaktov';
			SC_OvlHornychKontaktov.IdleTime.PT:= T#3s;
			SC_OvlHornychKontaktov.AlarmTime.PT:= T#6s;

			IF P4_FunkcnyTestA.Automat THEN
				SC_OvlHornychKontaktov.AlarmTime.IN:= TRUE;
			ELSE
				SC_OvlHornychKontaktov.IdleTime.IN:= TRUE;
			END_IF

			IF NOT SC_OvlHornychKontaktov.Switch1 THEN
				P4_FunkcnyTestA.OUT.HorneKontakty_VYSUN:= FALSE;
				P4_FunkcnyTestA.OUT.HorneKontakty_ZASUN:= TRUE;
				SC_OvlHornychKontaktov.Switch1:= TRUE;
			END_IF

			IF P4_FunkcnyTestA.IN.HorneKontakty_ZASUNUTE OR SC_OvlHornychKontaktov.IdleTime.Q THEN
				SC_OvlHornychKontaktov.ResetStep:= TRUE;
				SC_OvlHornychKontaktov.Step:= 0;
			ELSIF SC_OvlHornychKontaktov.AlarmTime.Q THEN
				P34_Alarmy[420]:= TRUE;
				P4_Pracovisko.STAV.Porucha_ST1:= TRUE;
			END_IF

	END_CASE

END_ACTION
```
